(* Logix 5000 project; controller reports 1756-L63 rev 20.11; software revision 20.04; part 38 of 52 *)

        [62].log_data[45].time := 3600.0, [62].log_data[45].valid := 1, [62].log_data[46].time := 3600.0, [62].log_data[46].valid := 1, [62].log_data[47].time := 3600.0, [62].log_data[47].valid := 1, [62].log_data[48].min := 6.623374, [62].log_data[48].max := 6.9811735, [62].log_data[48].total := 24355.637, [62].log_data[48].time := 3600.0, [62].log_data[48].minminute := 59, [62].log_data[48].maxminute := 38, [62].log_data[48].valid := 1, [62].log_data[49].min := 7.172454, [62].log_data[49].max := 9.684395, [62].log_data[49].total := 31171.475, [62].log_data[49].time := 3600.0, [62].log_data[49].minminute := 59, [62].log_data[49].maxminute := 34, [62].log_data[49].valid := 1, [62].log_data[50].min := 2.138653, [62].log_data[50].max := 2.2448862, [62].log_data[50].total := 7885.865, [62].log_data[50].time := 3600.0, [62].log_data[50].minminute := 33, [62].log_data[50].maxminute := 40, [62].log_data[50].valid := 1, [62].log_data[51].time := 3600.0, [62].log_data[51].valid := 1, [62].log_data[52].min := -2.880005, [62].log_data[52].max := 0.11999512, [62].log_data[52].total := -7701.21, [62].log_data[52].time := 3600.0, [62].log_data[52].minminute := 5, [62].log_data[52].maxminute := 3, [62].log_data[52].valid := 1, [62].log_data[53].min := -2.4800034, [62].log_data[53].max := 0.2400055, [62].log_data[53].total := -7366.718, [62].log_data[53].time := 3600.0, [62].log_data[53].maxminute := 40, [62].log_data[53].valid := 1, [62].log_data[54].max := 0.52250004, [62].log_data[54].total := 1217.2524, [62].log_data[54].time := 3600.0, [62].log_data[54].minminute := 3, [62].log_data[54].maxminute := 47, [62].log_data[54].valid := 1, [62].log_data[55].max := 0.5255, [62].log_data[55].total := 1254.6628, [62].log_data[55].time := 3600.0, [62].log_data[55].minminute := 7, [62].log_data[55].maxminute := 19, [62].log_data[55].valid := 1, [62].log_data[56].min := 0.15993154, [62].log_data[56].max := 0.16036338, [62].log_data[56].total := 576.5019, [62].log_data[56].time := 3600.0, [62].log_data[56].minminute := 1, [62].log_data[56].maxminute := 9,
        [62].log_data[56].valid := 1, [62].log_data[57].min := 0.26655704, [62].log_data[57].max := 0.26718515, [62].log_data[57].total := 960.41205, [62].log_data[57].time := 3600.0, [62].log_data[57].minminute := 32, [62].log_data[57].valid := 1, [62].log_data[58].time := 3600.0, [62].log_data[58].valid := 1, [62].log_data[59].time := 3600.0, [62].log_data[59].valid := 1, [62].log_data[60].valid := 1, [62].log_data[61].valid := 1, [62].log_data[62].valid := 1, [62].log_data[63].valid := 1, [62].log_data[64].valid := 1, [62].log_data[65].valid := 1, [62].log_data[66].valid := 1, [62].log_data[67].valid := 1, [62].log_data[68].valid := 1, [62].log_data[69].valid := 1, [62].log_data[70].valid := 1, [62].log_data[71].valid := 1, [62].log_data[72].valid := 1, [62].log_data[73].valid := 1, [62].log_data[74].valid := 1, [62].log_data[75].valid := 1, [62].log_data[76].valid := 1, [62].log_data[77].valid := 1, [62].log_data[78].valid := 1, [62].log_data[79].valid := 1, [62].log_data[80].valid := 1, [62].log_data[81].valid := 1, [62].log_data[82].valid := 1, [62].log_data[83].valid := 1, [62].log_data[84].valid := 1, [62].log_data[85].valid := 1, [62].log_data[86].valid := 1, [62].log_data[87].valid := 1, [62].log_data[88].valid := 1, [62].log_data[89].valid := 1, [62].log_data[90].valid := 1, [62].log_data[91].valid := 1, [62].log_data[92].valid := 1, [62].log_data[93].valid := 1, [62].log_data[94].valid := 1, [62].log_data[95].valid := 1, [62].log_data[96].valid := 1, [62].log_data[97].valid := 1, [62].log_data[98].valid := 1, [62].log_data[99].valid := 1, [62].log_data[100].valid := 1, [62].log_data[101].valid := 1, [62].log_data[102].valid := 1, [62].log_data[103].valid := 1, [62].log_data[104].valid := 1, [62].log_data[105].valid := 1, [62].log_data[106].valid := 1, [62].log_data[107].valid := 1, [62].log_data[108].valid := 1,
        [62].log_data[109].valid := 1, [62].log_data[110].valid := 1, [62].log_data[111].valid := 1, [62].log_data[112].valid := 1, [62].log_data[113].valid := 1, [62].log_data[114].valid := 1, [62].log_data[115].valid := 1, [62].log_data[116].valid := 1, [62].log_data[117].valid := 1, [62].log_data[118].valid := 1, [62].log_data[119].valid := 1, [62].log_data[120].valid := 1, [62].log_data[121].valid := 1, [62].log_data[122].valid := 1, [62].log_data[123].valid := 1, [62].log_data[124].valid := 1, [62].time.Year := 2023, [62].time.Month := 1, [62].time.Day := 15, [62].time.Hour := 17, [62].time.Minute := 59, [62].time.Second := 59, [63].log_data[0].min := 1.0, [63].log_data[0].max := 1.0, [63].log_data[0].total := 3600.0, [63].log_data[0].time := 3600.0, [63].log_data[0].valid := 1, [63].log_data[1].time := 3600.0, [63].log_data[1].valid := 1, [63].log_data[2].time := 3600.0, [63].log_data[2].valid := 1, [63].log_data[3].time := 3600.0, [63].log_data[3].valid := 1, [63].log_data[4].time := 3600.0, [63].log_data[4].valid := 1, [63].log_data[5].time := 3600.0, [63].log_data[5].valid := 1, [63].log_data[6].time := 3600.0, [63].log_data[6].valid := 1, [63].log_data[7].time := 3600.0, [63].log_data[7].valid := 1, [63].log_data[8].min := 1.0, [63].log_data[8].max := 1.0, [63].log_data[8].total := 3600.0, [63].log_data[8].time := 3600.0, [63].log_data[8].valid := 1, [63].log_data[9].min := 1.0, [63].log_data[9].max := 1.0, [63].log_data[9].total := 3600.0, [63].log_data[9].time := 3600.0, [63].log_data[9].valid := 1, [63].log_data[10].min := 1.0, [63].log_data[10].max := 1.0, [63].log_data[10].total := 3600.0, [63].log_data[10].time := 3600.0, [63].log_data[10].valid := 1, [63].log_data[11].time := 3600.0, [63].log_data[11].valid := 1, [63].log_data[12].min := 1.0, [63].log_data[12].max := 1.0,
        [63].log_data[12].total := 3600.0, [63].log_data[12].time := 3600.0, [63].log_data[12].valid := 1, [63].log_data[13].min := 1.0, [63].log_data[13].max := 1.0, [63].log_data[13].total := 3600.0, [63].log_data[13].time := 3600.0, [63].log_data[13].valid := 1, [63].log_data[14].time := 3600.0, [63].log_data[14].valid := 1, [63].log_data[15].time := 3600.0, [63].log_data[15].valid := 1, [63].log_data[16].time := 3600.0, [63].log_data[16].valid := 1, [63].log_data[17].min := 1.0, [63].log_data[17].max := 1.0, [63].log_data[17].total := 3600.0, [63].log_data[17].time := 3600.0, [63].log_data[17].valid := 1, [63].log_data[18].time := 3600.0, [63].log_data[18].valid := 1, [63].log_data[19].time := 3600.0, [63].log_data[19].valid := 1, [63].log_data[20].time := 3600.0, [63].log_data[20].valid := 1, [63].log_data[21].min := 1.0, [63].log_data[21].max := 1.0, [63].log_data[21].total := 3600.0, [63].log_data[21].time := 3600.0, [63].log_data[21].valid := 1, [63].log_data[22].time := 3600.0, [63].log_data[22].valid := 1, [63].log_data[23].time := 3600.0, [63].log_data[23].valid := 1, [63].log_data[24].time := 3600.0, [63].log_data[24].valid := 1, [63].log_data[25].time := 3600.0, [63].log_data[25].valid := 1, [63].log_data[26].time := 3600.0, [63].log_data[26].valid := 1, [63].log_data[27].time := 3600.0, [63].log_data[27].valid := 1, [63].log_data[28].time := 3600.0, [63].log_data[28].valid := 1, [63].log_data[29].min := 1.0, [63].log_data[29].max := 1.0, [63].log_data[29].total := 3600.0, [63].log_data[29].time := 3600.0, [63].log_data[29].valid := 1, [63].log_data[30].min := 1.0, [63].log_data[30].max := 1.0, [63].log_data[30].total := 3600.0, [63].log_data[30].time := 3600.0, [63].log_data[30].valid := 1, [63].log_data[31].max := 1.0, [63].log_data[31].total := 1629.998, [63].log_data[31].time := 3600.0, [63].log_data[31].maxminute := 8, [63].log_data[31].valid := 1, [63].log_data[32].max := 1.0,
        [63].log_data[32].total := 1502.498, [63].log_data[32].time := 3600.0, [63].log_data[32].minminute := 6, [63].log_data[32].valid := 1, [63].log_data[33].time := 3600.0, [63].log_data[33].valid := 1, [63].log_data[34].time := 3600.0, [63].log_data[34].valid := 1, [63].log_data[35].max := 1.0, [63].log_data[35].total := 1440.7471, [63].log_data[35].time := 3600.0, [63].log_data[35].valid := 1, [63].log_data[36].max := 1.0, [63].log_data[36].total := 1629.7471, [63].log_data[36].time := 3600.0, [63].log_data[36].maxminute := 1, [63].log_data[36].valid := 1, [63].log_data[37].time := 3600.0, [63].log_data[37].valid := 1, [63].log_data[38].time := 3600.0, [63].log_data[38].valid := 1, [63].log_data[39].min := 0.99965274, [63].log_data[39].max := 1.0098991, [63].log_data[39].total := 3618.9036, [63].log_data[39].time := 3600.0, [63].log_data[39].minminute := 27, [63].log_data[39].maxminute := 51, [63].log_data[39].valid := 1, [63].log_data[40].min := 7.5689883, [63].log_data[40].max := 7.599217, [63].log_data[40].total := 27323.691, [63].log_data[40].time := 3600.0, [63].log_data[40].minminute := 52, [63].log_data[40].maxminute := 29, [63].log_data[40].valid := 1, [63].log_data[41].min := 0.02273633, [63].log_data[41].max := 0.03628052, [63].log_data[41].total := 100.63758, [63].log_data[41].time := 3600.0, [63].log_data[41].minminute := 33, [63].log_data[41].maxminute := 10, [63].log_data[41].valid := 1, [63].log_data[42].min := 2.2918782, [63].log_data[42].max := 2.2965894, [63].log_data[42].total := 8260.206, [63].log_data[42].time := 3600.0, [63].log_data[42].minminute := 14, [63].log_data[42].maxminute := 40, [63].log_data[42].valid := 1, [63].log_data[43].min := -0.27999878, [63].log_data[43].max := -0.27999878, [63].log_data[43].total := -1007.8613, [63].log_data[43].time := 3600.0, [63].log_data[43].valid := 1, [63].log_data[44].min := -0.3199997, [63].log_data[44].max := -0.30000305, [63].log_data[44].total := -1092.1874, [63].log_data[44].time := 3600.0, [63].log_data[44].valid := 1, [63].log_data[45].time := 3600.0,
        [63].log_data[45].valid := 1, [63].log_data[46].time := 3600.0, [63].log_data[46].valid := 1, [63].log_data[47].time := 3600.0, [63].log_data[47].valid := 1, [63].log_data[48].min := 6.590947, [63].log_data[48].max := 6.7857857, [63].log_data[48].total := 24242.467, [63].log_data[48].time := 3600.0, [63].log_data[48].minminute := 6, [63].log_data[48].maxminute := 19, [63].log_data[48].valid := 1, [63].log_data[49].min := 7.1553764, [63].log_data[49].max := 9.774297, [63].log_data[49].total := 32409.39, [63].log_data[49].time := 3600.0, [63].log_data[49].maxminute := 58, [63].log_data[49].valid := 1, [63].log_data[50].min := 2.1388886, [63].log_data[50].max := 2.2252176, [63].log_data[50].total := 7860.6226, [63].log_data[50].time := 3600.0, [63].log_data[50].minminute := 59, [63].log_data[50].valid := 1, [63].log_data[51].time := 3600.0, [63].log_data[51].valid := 1, [63].log_data[52].min := -2.9000015, [63].log_data[52].max := 0.11999512, [63].log_data[52].total := -7927.2964, [63].log_data[52].time := 3600.0, [63].log_data[52].minminute := 8, [63].log_data[52].maxminute := 7, [63].log_data[52].valid := 1, [63].log_data[53].min := -2.5, [63].log_data[53].max := 0.27999878, [63].log_data[53].total := -7180.0005, [63].log_data[53].time := 3600.0, [63].log_data[53].minminute := 13, [63].log_data[53].maxminute := 1, [63].log_data[53].valid := 1, [63].log_data[54].max := 0.531, [63].log_data[54].total := 1244.2853, [63].log_data[54].time := 3600.0, [63].log_data[54].minminute := 6, [63].log_data[54].maxminute := 29, [63].log_data[54].valid := 1, [63].log_data[55].max := 0.5185, [63].log_data[55].total := 1217.0046, [63].log_data[55].time := 3600.0, [63].log_data[55].maxminute := 54, [63].log_data[55].valid := 1, [63].log_data[56].min := 0.1599708, [63].log_data[56].max := 0.16040264, [63].log_data[56].total := 576.58856, [63].log_data[56].time := 3600.0, [63].log_data[56].minminute := 11, [63].log_data[56].maxminute := 26, [63].log_data[56].valid := 1, [63].log_data[57].min := 0.26534003, [63].log_data[57].max := 0.26694962,
        [63].log_data[57].total := 956.40753, [63].log_data[57].time := 3600.0, [63].log_data[57].minminute := 15, [63].log_data[57].valid := 1, [63].log_data[58].time := 3600.0, [63].log_data[58].valid := 1, [63].log_data[59].time := 3600.0, [63].log_data[59].valid := 1, [63].log_data[60].valid := 1, [63].log_data[61].valid := 1, [63].log_data[62].valid := 1, [63].log_data[63].valid := 1, [63].log_data[64].valid := 1, [63].log_data[65].valid := 1, [63].log_data[66].valid := 1, [63].log_data[67].valid := 1, [63].log_data[68].valid := 1, [63].log_data[69].valid := 1, [63].log_data[70].valid := 1, [63].log_data[71].valid := 1, [63].log_data[72].valid := 1, [63].log_data[73].valid := 1, [63].log_data[74].valid := 1, [63].log_data[75].valid := 1, [63].log_data[76].valid := 1, [63].log_data[77].valid := 1, [63].log_data[78].valid := 1, [63].log_data[79].valid := 1, [63].log_data[80].valid := 1, [63].log_data[81].valid := 1, [63].log_data[82].valid := 1, [63].log_data[83].valid := 1, [63].log_data[84].valid := 1, [63].log_data[85].valid := 1, [63].log_data[86].valid := 1, [63].log_data[87].valid := 1, [63].log_data[88].valid := 1, [63].log_data[89].valid := 1, [63].log_data[90].valid := 1, [63].log_data[91].valid := 1, [63].log_data[92].valid := 1, [63].log_data[93].valid := 1, [63].log_data[94].valid := 1, [63].log_data[95].valid := 1, [63].log_data[96].valid := 1, [63].log_data[97].valid := 1, [63].log_data[98].valid := 1, [63].log_data[99].valid := 1, [63].log_data[100].valid := 1, [63].log_data[101].valid := 1, [63].log_data[102].valid := 1, [63].log_data[103].valid := 1, [63].log_data[104].valid := 1, [63].log_data[105].valid := 1, [63].log_data[106].valid := 1, [63].log_data[107].valid := 1, [63].log_data[108].valid := 1, [63].log_data[109].valid := 1, [63].log_data[110].valid := 1, [63].log_data[111].valid := 1,
        [63].log_data[112].valid := 1, [63].log_data[113].valid := 1, [63].log_data[114].valid := 1, [63].log_data[115].valid := 1, [63].log_data[116].valid := 1, [63].log_data[117].valid := 1, [63].log_data[118].valid := 1, [63].log_data[119].valid := 1, [63].log_data[120].valid := 1, [63].log_data[121].valid := 1, [63].log_data[122].valid := 1, [63].log_data[123].valid := 1, [63].log_data[124].valid := 1, [63].time.Year := 2023, [63].time.Month := 1, [63].time.Day := 15, [63].time.Hour := 18, [63].time.Minute := 59, [63].time.Second := 59, [64].log_data[0].min := 1.0, [64].log_data[0].max := 1.0, [64].log_data[0].total := 3600.0, [64].log_data[0].time := 3600.0, [64].log_data[0].valid := 1, [64].log_data[1].max := 1.0, [64].log_data[1].total := 575.0, [64].log_data[1].time := 3600.0, [64].log_data[1].valid := 1, [64].log_data[2].max := 1.0, [64].log_data[2].total := 571.5, [64].log_data[2].time := 3600.0, [64].log_data[2].valid := 1, [64].log_data[3].time := 3600.0, [64].log_data[3].valid := 1, [64].log_data[4].time := 3600.0, [64].log_data[4].valid := 1, [64].log_data[5].max := 1.0, [64].log_data[5].total := 239.5, [64].log_data[5].time := 3600.0, [64].log_data[5].maxminute := 2, [64].log_data[5].valid := 1, [64].log_data[6].time := 3600.0, [64].log_data[6].valid := 1, [64].log_data[7].time := 3600.0, [64].log_data[7].valid := 1, [64].log_data[8].min := 1.0, [64].log_data[8].max := 1.0, [64].log_data[8].total := 3600.0, [64].log_data[8].time := 3600.0, [64].log_data[8].valid := 1, [64].log_data[9].min := 1.0, [64].log_data[9].max := 1.0, [64].log_data[9].total := 3600.0, [64].log_data[9].time := 3600.0, [64].log_data[9].valid := 1, [64].log_data[10].min := 1.0, [64].log_data[10].max := 1.0, [64].log_data[10].total := 3600.0, [64].log_data[10].time := 3600.0, [64].log_data[10].valid := 1,
        [64].log_data[11].time := 3600.0, [64].log_data[11].valid := 1, [64].log_data[12].min := 1.0, [64].log_data[12].max := 1.0, [64].log_data[12].total := 3600.0, [64].log_data[12].time := 3600.0, [64].log_data[12].valid := 1, [64].log_data[13].min := 1.0, [64].log_data[13].max := 1.0, [64].log_data[13].total := 3600.0, [64].log_data[13].time := 3600.0, [64].log_data[13].valid := 1, [64].log_data[14].time := 3600.0, [64].log_data[14].valid := 1, [64].log_data[15].time := 3600.0, [64].log_data[15].valid := 1, [64].log_data[16].time := 3600.0, [64].log_data[16].valid := 1, [64].log_data[17].min := 1.0, [64].log_data[17].max := 1.0, [64].log_data[17].total := 3600.0, [64].log_data[17].time := 3600.0, [64].log_data[17].valid := 1, [64].log_data[18].time := 3600.0, [64].log_data[18].valid := 1, [64].log_data[19].time := 3600.0, [64].log_data[19].valid := 1, [64].log_data[20].time := 3600.0, [64].log_data[20].valid := 1, [64].log_data[21].min := 1.0, [64].log_data[21].max := 1.0, [64].log_data[21].total := 3600.0, [64].log_data[21].time := 3600.0, [64].log_data[21].valid := 1, [64].log_data[22].time := 3600.0, [64].log_data[22].valid := 1, [64].log_data[23].time := 3600.0, [64].log_data[23].valid := 1, [64].log_data[24].time := 3600.0, [64].log_data[24].valid := 1, [64].log_data[25].time := 3600.0, [64].log_data[25].valid := 1, [64].log_data[26].time := 3600.0, [64].log_data[26].valid := 1, [64].log_data[27].time := 3600.0, [64].log_data[27].valid := 1, [64].log_data[28].time := 3600.0, [64].log_data[28].valid := 1, [64].log_data[29].min := 1.0, [64].log_data[29].max := 1.0, [64].log_data[29].total := 3600.0, [64].log_data[29].time := 3600.0, [64].log_data[29].valid := 1, [64].log_data[30].min := 1.0, [64].log_data[30].max := 1.0, [64].log_data[30].total := 3600.0, [64].log_data[30].time := 3600.0, [64].log_data[30].valid := 1, [64].log_data[31].max := 1.0, [64].log_data[31].total := 1467.2471,
        [64].log_data[31].time := 3600.0, [64].log_data[31].maxminute := 11, [64].log_data[31].valid := 1, [64].log_data[32].max := 1.0, [64].log_data[32].total := 1629.7471, [64].log_data[32].time := 3600.0, [64].log_data[32].maxminute := 1, [64].log_data[32].valid := 1, [64].log_data[33].time := 3600.0, [64].log_data[33].valid := 1, [64].log_data[34].time := 3600.0, [64].log_data[34].valid := 1, [64].log_data[35].max := 1.0, [64].log_data[35].total := 1440.7471, [64].log_data[35].time := 3600.0, [64].log_data[35].minminute := 3, [64].log_data[35].valid := 1, [64].log_data[36].max := 1.0, [64].log_data[36].total := 1629.7471, [64].log_data[36].time := 3600.0, [64].log_data[36].maxminute := 5, [64].log_data[36].valid := 1, [64].log_data[37].max := 7.22856, [64].log_data[37].total := 3622.7856, [64].log_data[37].time := 3600.0, [64].log_data[37].maxminute := 1, [64].log_data[37].valid := 1, [64].log_data[38].time := 3600.0, [64].log_data[38].valid := 1, [64].log_data[39].min := 0.9982394, [64].log_data[39].max := 1.02203, [64].log_data[39].total := 3625.5354, [64].log_data[39].time := 3600.0, [64].log_data[39].minminute := 8, [64].log_data[39].maxminute := 6, [64].log_data[39].valid := 1, [64].log_data[40].min := 7.560194, [64].log_data[40].max := 7.6063623, [64].log_data[40].total := 27324.1, [64].log_data[40].time := 3600.0, [64].log_data[40].minminute := 56, [64].log_data[40].maxminute := 59, [64].log_data[40].valid := 1, [64].log_data[41].min := 0.025877198, [64].log_data[41].max := 0.044524662, [64].log_data[41].total := 125.660706, [64].log_data[41].time := 3600.0, [64].log_data[41].maxminute := 30, [64].log_data[41].valid := 1, [64].log_data[42].min := 2.2917604, [64].log_data[42].max := 2.2964714, [64].log_data[42].total := 8260.182, [64].log_data[42].time := 3600.0, [64].log_data[42].minminute := 28, [64].log_data[42].maxminute := 24, [64].log_data[42].valid := 1, [64].log_data[43].min := -0.27999878, [64].log_data[43].max := -0.26000214, [64].log_data[43].total := -1007.73706, [64].log_data[43].time := 3600.0,
        [64].log_data[43].maxminute := 9, [64].log_data[43].valid := 1, [64].log_data[44].min := -0.3199997, [64].log_data[44].max := -0.30000305, [64].log_data[44].total := -1087.6062, [64].log_data[44].time := 3600.0, [64].log_data[44].valid := 1, [64].log_data[45].time := 3600.0, [64].log_data[45].valid := 1, [64].log_data[46].time := 3600.0, [64].log_data[46].valid := 1, [64].log_data[47].time := 3600.0, [64].log_data[47].valid := 1, [64].log_data[48].min := 6.588199, [64].log_data[48].max := 6.952594, [64].log_data[48].total := 24228.959, [64].log_data[48].time := 3600.0, [64].log_data[48].minminute := 33, [64].log_data[48].maxminute := 3, [64].log_data[48].valid := 1, [64].log_data[49].min := 7.1818757, [64].log_data[49].max := 9.775277, [64].log_data[49].total := 29847.389, [64].log_data[49].time := 3600.0, [64].log_data[49].minminute := 30, [64].log_data[49].maxminute := 1, [64].log_data[49].valid := 1, [64].log_data[50].min := 2.13512, [64].log_data[50].max := 2.2438262, [64].log_data[50].total := 7948.6934, [64].log_data[50].time := 3600.0, [64].log_data[50].minminute := 1, [64].log_data[50].maxminute := 11, [64].log_data[50].valid := 1, [64].log_data[51].time := 3600.0, [64].log_data[51].valid := 1, [64].log_data[52].min := -2.959999, [64].log_data[52].max := 0.11999512, [64].log_data[52].total := -7812.1035, [64].log_data[52].time := 3600.0, [64].log_data[52].minminute := 11, [64].log_data[52].valid := 1, [64].log_data[53].min := -2.600006, [64].log_data[53].max := 0.2400055, [64].log_data[53].total := -7210.3994, [64].log_data[53].time := 3600.0, [64].log_data[53].minminute := 15, [64].log_data[53].maxminute := 25, [64].log_data[53].valid := 1, [64].log_data[54].max := 0.54, [64].log_data[54].total := 1227.2667, [64].log_data[54].time := 3600.0, [64].log_data[54].maxminute := 11, [64].log_data[54].valid := 1, [64].log_data[55].max := 0.539, [64].log_data[55].total := 1217.0822, [64].log_data[55].time := 3600.0, [64].log_data[55].minminute := 3, [64].log_data[55].maxminute := 57, [64].log_data[55].valid := 1,
        [64].log_data[56].min := 0.16001005, [64].log_data[56].max := 0.16044189, [64].log_data[56].total := 576.6807, [64].log_data[56].time := 3600.0, [64].log_data[56].minminute := 32, [64].log_data[56].maxminute := 29, [64].log_data[56].valid := 1, [64].log_data[57].min := 0.26380894, [64].log_data[57].max := 0.26569337, [64].log_data[57].total := 953.66, [64].log_data[57].time := 3600.0, [64].log_data[57].minminute := 50, [64].log_data[57].maxminute := 6, [64].log_data[57].valid := 1, [64].log_data[58].time := 3600.0, [64].log_data[58].valid := 1, [64].log_data[59].time := 3600.0, [64].log_data[59].valid := 1, [64].log_data[60].valid := 1, [64].log_data[61].valid := 1, [64].log_data[62].valid := 1, [64].log_data[63].valid := 1, [64].log_data[64].valid := 1, [64].log_data[65].valid := 1, [64].log_data[66].valid := 1, [64].log_data[67].valid := 1, [64].log_data[68].valid := 1, [64].log_data[69].valid := 1, [64].log_data[70].valid := 1, [64].log_data[71].valid := 1, [64].log_data[72].valid := 1, [64].log_data[73].valid := 1, [64].log_data[74].valid := 1, [64].log_data[75].valid := 1, [64].log_data[76].valid := 1, [64].log_data[77].valid := 1, [64].log_data[78].valid := 1, [64].log_data[79].valid := 1, [64].log_data[80].valid := 1, [64].log_data[81].valid := 1, [64].log_data[82].valid := 1, [64].log_data[83].valid := 1, [64].log_data[84].valid := 1, [64].log_data[85].valid := 1, [64].log_data[86].valid := 1, [64].log_data[87].valid := 1, [64].log_data[88].valid := 1, [64].log_data[89].valid := 1, [64].log_data[90].valid := 1, [64].log_data[91].valid := 1, [64].log_data[92].valid := 1, [64].log_data[93].valid := 1, [64].log_data[94].valid := 1, [64].log_data[95].valid := 1, [64].log_data[96].valid := 1, [64].log_data[97].valid := 1, [64].log_data[98].valid := 1, [64].log_data[99].valid := 1, [64].log_data[100].valid := 1, [64].log_data[101].valid := 1,
        [64].log_data[102].valid := 1, [64].log_data[103].valid := 1, [64].log_data[104].valid := 1, [64].log_data[105].valid := 1, [64].log_data[106].valid := 1, [64].log_data[107].valid := 1, [64].log_data[108].valid := 1, [64].log_data[109].valid := 1, [64].log_data[110].valid := 1, [64].log_data[111].valid := 1, [64].log_data[112].valid := 1, [64].log_data[113].valid := 1, [64].log_data[114].valid := 1, [64].log_data[115].valid := 1, [64].log_data[116].valid := 1, [64].log_data[117].valid := 1, [64].log_data[118].valid := 1, [64].log_data[119].valid := 1, [64].log_data[120].valid := 1, [64].log_data[121].valid := 1, [64].log_data[122].valid := 1, [64].log_data[123].valid := 1, [64].log_data[124].valid := 1, [64].time.Year := 2023, [64].time.Month := 1, [64].time.Day := 15, [64].time.Hour := 19, [64].time.Minute := 59, [64].time.Second := 59, [65].log_data[0].min := 1.0, [65].log_data[0].max := 1.0, [65].log_data[0].total := 3600.0, [65].log_data[0].time := 3600.0, [65].log_data[0].valid := 1, [65].log_data[1].max := 1.0, [65].log_data[1].total := 552.0, [65].log_data[1].time := 3600.0, [65].log_data[1].maxminute := 8, [65].log_data[1].valid := 1, [65].log_data[2].max := 1.0, [65].log_data[2].total := 548.5, [65].log_data[2].time := 3600.0, [65].log_data[2].maxminute := 8, [65].log_data[2].valid := 1, [65].log_data[3].time := 3600.0, [65].log_data[3].valid := 1, [65].log_data[4].time := 3600.0, [65].log_data[4].valid := 1, [65].log_data[5].max := 1.0, [65].log_data[5].total := 250.5, [65].log_data[5].time := 3600.0, [65].log_data[5].maxminute := 10, [65].log_data[5].valid := 1, [65].log_data[6].time := 3600.0, [65].log_data[6].valid := 1, [65].log_data[7].time := 3600.0, [65].log_data[7].valid := 1, [65].log_data[8].min := 1.0, [65].log_data[8].max := 1.0, [65].log_data[8].total := 3600.0,
        [65].log_data[8].time := 3600.0, [65].log_data[8].valid := 1, [65].log_data[9].min := 1.0, [65].log_data[9].max := 1.0, [65].log_data[9].total := 3600.0, [65].log_data[9].time := 3600.0, [65].log_data[9].valid := 1, [65].log_data[10].min := 1.0, [65].log_data[10].max := 1.0, [65].log_data[10].total := 3600.0, [65].log_data[10].time := 3600.0, [65].log_data[10].valid := 1, [65].log_data[11].time := 3600.0, [65].log_data[11].valid := 1, [65].log_data[12].min := 1.0, [65].log_data[12].max := 1.0, [65].log_data[12].total := 3600.0, [65].log_data[12].time := 3600.0, [65].log_data[12].valid := 1, [65].log_data[13].min := 1.0, [65].log_data[13].max := 1.0, [65].log_data[13].total := 3600.0, [65].log_data[13].time := 3600.0, [65].log_data[13].valid := 1, [65].log_data[14].time := 3600.0, [65].log_data[14].valid := 1, [65].log_data[15].time := 3600.0, [65].log_data[15].valid := 1, [65].log_data[16].time := 3600.0, [65].log_data[16].valid := 1, [65].log_data[17].min := 1.0, [65].log_data[17].max := 1.0, [65].log_data[17].total := 3600.0, [65].log_data[17].time := 3600.0, [65].log_data[17].valid := 1, [65].log_data[18].time := 3600.0, [65].log_data[18].valid := 1, [65].log_data[19].time := 3600.0, [65].log_data[19].valid := 1, [65].log_data[20].time := 3600.0, [65].log_data[20].valid := 1, [65].log_data[21].min := 1.0, [65].log_data[21].max := 1.0, [65].log_data[21].total := 3600.0, [65].log_data[21].time := 3600.0, [65].log_data[21].valid := 1, [65].log_data[22].time := 3600.0, [65].log_data[22].valid := 1, [65].log_data[23].time := 3600.0, [65].log_data[23].valid := 1, [65].log_data[24].time := 3600.0, [65].log_data[24].valid := 1, [65].log_data[25].time := 3600.0, [65].log_data[25].valid := 1, [65].log_data[26].time := 3600.0, [65].log_data[26].valid := 1, [65].log_data[27].time := 3600.0, [65].log_data[27].valid := 1, [65].log_data[28].time := 3600.0, [65].log_data[28].valid := 1,
        [65].log_data[29].min := 1.0, [65].log_data[29].max := 1.0, [65].log_data[29].total := 3600.0, [65].log_data[29].time := 3600.0, [65].log_data[29].valid := 1, [65].log_data[30].min := 1.0, [65].log_data[30].max := 1.0, [65].log_data[30].total := 3600.0, [65].log_data[30].time := 3600.0, [65].log_data[30].valid := 1, [65].log_data[31].max := 1.0, [65].log_data[31].total := 1441.249, [65].log_data[31].time := 3600.0, [65].log_data[31].minminute := 2, [65].log_data[31].valid := 1, [65].log_data[32].max := 1.0, [65].log_data[32].total := 1629.749, [65].log_data[32].time := 3600.0, [65].log_data[32].maxminute := 4, [65].log_data[32].valid := 1, [65].log_data[33].time := 3600.0, [65].log_data[33].valid := 1, [65].log_data[34].time := 3600.0, [65].log_data[34].valid := 1, [65].log_data[35].max := 1.0, [65].log_data[35].total := 1491.998, [65].log_data[35].time := 3600.0, [65].log_data[35].minminute := 6, [65].log_data[35].valid := 1, [65].log_data[36].max := 1.0, [65].log_data[36].total := 1629.998, [65].log_data[36].time := 3600.0, [65].log_data[36].maxminute := 8, [65].log_data[36].valid := 1, [65].log_data[37].max := 7.450369, [65].log_data[37].total := 3580.0767, [65].log_data[37].time := 3600.0, [65].log_data[37].maxminute := 9, [65].log_data[37].valid := 1, [65].log_data[38].time := 3600.0, [65].log_data[38].valid := 1, [65].log_data[39].min := 0.99800396, [65].log_data[39].max := 1.0223833, [65].log_data[39].total := 3620.6714, [65].log_data[39].time := 3600.0, [65].log_data[39].minminute := 59, [65].log_data[39].maxminute := 10, [65].log_data[39].valid := 1, [65].log_data[40].min := 7.557446, [65].log_data[40].max := 7.611859, [65].log_data[40].total := 27325.555, [65].log_data[40].time := 3600.0, [65].log_data[40].minminute := 37, [65].log_data[40].maxminute := 40, [65].log_data[40].valid := 1, [65].log_data[41].min := 0.02273633, [65].log_data[41].max := 0.034317628, [65].log_data[41].total := 96.31372, [65].log_data[41].time := 3600.0, [65].log_data[41].minminute := 29,
        [65].log_data[41].maxminute := 7, [65].log_data[41].valid := 1, [65].log_data[42].min := 2.291996, [65].log_data[42].max := 2.2968247, [65].log_data[42].total := 8260.134, [65].log_data[42].time := 3600.0, [65].log_data[42].minminute := 40, [65].log_data[42].maxminute := 35, [65].log_data[42].valid := 1, [65].log_data[43].min := -0.27999878, [65].log_data[43].max := -0.26000214, [65].log_data[43].total := -1007.21295, [65].log_data[43].time := 3600.0, [65].log_data[43].maxminute := 9, [65].log_data[43].valid := 1, [65].log_data[44].min := -0.3199997, [65].log_data[44].max := -0.30000305, [65].log_data[44].total := -1082.1633, [65].log_data[44].time := 3600.0, [65].log_data[44].valid := 1, [65].log_data[45].time := 3600.0, [65].log_data[45].valid := 1, [65].log_data[46].time := 3600.0, [65].log_data[46].valid := 1, [65].log_data[47].time := 3600.0, [65].log_data[47].valid := 1, [65].log_data[48].min := 6.5824285, [65].log_data[48].max := 6.969357, [65].log_data[48].total := 24224.227, [65].log_data[48].time := 3600.0, [65].log_data[48].minminute := 42, [65].log_data[48].maxminute := 17, [65].log_data[48].valid := 1, [65].log_data[49].min := 7.0841227, [65].log_data[49].max := 9.659073, [65].log_data[49].total := 29661.438, [65].log_data[49].time := 3600.0, [65].log_data[49].minminute := 39, [65].log_data[49].maxminute := 10, [65].log_data[49].valid := 1, [65].log_data[50].min := 2.163268, [65].log_data[50].max := 2.276332, [65].log_data[50].total := 8044.48, [65].log_data[50].time := 3600.0, [65].log_data[50].minminute := 10, [65].log_data[50].maxminute := 18, [65].log_data[50].valid := 1, [65].log_data[51].time := 3600.0, [65].log_data[51].valid := 1, [65].log_data[52].min := -2.959999, [65].log_data[52].max := 0.11999512, [65].log_data[52].total := -7730.7188, [65].log_data[52].time := 3600.0, [65].log_data[52].minminute := 56, [65].log_data[52].maxminute := 2, [65].log_data[52].valid := 1, [65].log_data[53].min := -2.6600037, [65].log_data[53].max := 0.27999878, [65].log_data[53].total := -7362.1255, [65].log_data[53].time := 3600.0,
        [65].log_data[53].minminute := 8, [65].log_data[53].maxminute := 7, [65].log_data[53].valid := 1, [65].log_data[54].max := 0.53, [65].log_data[54].total := 1217.8265, [65].log_data[54].time := 3600.0, [65].log_data[54].minminute := 2, [65].log_data[54].maxminute := 56, [65].log_data[54].valid := 1, [65].log_data[55].max := 0.546, [65].log_data[55].total := 1240.171, [65].log_data[55].time := 3600.0, [65].log_data[55].minminute := 6, [65].log_data[55].maxminute := 18, [65].log_data[55].valid := 1, [65].log_data[56].min := 0.16001005, [65].log_data[56].max := 0.16044189, [65].log_data[56].total := 576.7335, [65].log_data[56].time := 3600.0, [65].log_data[56].minminute := 39, [65].log_data[56].maxminute := 14, [65].log_data[56].valid := 1, [65].log_data[57].min := 0.2618068, [65].log_data[57].max := 0.26424077, [65].log_data[57].total := 948.47955, [65].log_data[57].time := 3600.0, [65].log_data[57].minminute := 58, [65].log_data[57].maxminute := 13, [65].log_data[57].valid := 1, [65].log_data[58].time := 3600.0, [65].log_data[58].valid := 1, [65].log_data[59].time := 3600.0, [65].log_data[59].valid := 1, [65].log_data[60].valid := 1, [65].log_data[61].valid := 1, [65].log_data[62].valid := 1, [65].log_data[63].valid := 1, [65].log_data[64].valid := 1, [65].log_data[65].valid := 1, [65].log_data[66].valid := 1, [65].log_data[67].valid := 1, [65].log_data[68].valid := 1, [65].log_data[69].valid := 1, [65].log_data[70].valid := 1, [65].log_data[71].valid := 1, [65].log_data[72].valid := 1, [65].log_data[73].valid := 1, [65].log_data[74].valid := 1, [65].log_data[75].valid := 1, [65].log_data[76].valid := 1, [65].log_data[77].valid := 1, [65].log_data[78].valid := 1, [65].log_data[79].valid := 1, [65].log_data[80].valid := 1, [65].log_data[81].valid := 1, [65].log_data[82].valid := 1, [65].log_data[83].valid := 1, [65].log_data[84].valid := 1, [65].log_data[85].valid := 1, [65].log_data[86].valid := 1,
        [65].log_data[87].valid := 1, [65].log_data[88].valid := 1, [65].log_data[89].valid := 1, [65].log_data[90].valid := 1, [65].log_data[91].valid := 1, [65].log_data[92].valid := 1, [65].log_data[93].valid := 1, [65].log_data[94].valid := 1, [65].log_data[95].valid := 1, [65].log_data[96].valid := 1, [65].log_data[97].valid := 1, [65].log_data[98].valid := 1, [65].log_data[99].valid := 1, [65].log_data[100].valid := 1, [65].log_data[101].valid := 1, [65].log_data[102].valid := 1, [65].log_data[103].valid := 1, [65].log_data[104].valid := 1, [65].log_data[105].valid := 1, [65].log_data[106].valid := 1, [65].log_data[107].valid := 1, [65].log_data[108].valid := 1, [65].log_data[109].valid := 1, [65].log_data[110].valid := 1, [65].log_data[111].valid := 1, [65].log_data[112].valid := 1, [65].log_data[113].valid := 1, [65].log_data[114].valid := 1, [65].log_data[115].valid := 1, [65].log_data[116].valid := 1, [65].log_data[117].valid := 1, [65].log_data[118].valid := 1, [65].log_data[119].valid := 1, [65].log_data[120].valid := 1, [65].log_data[121].valid := 1, [65].log_data[122].valid := 1, [65].log_data[123].valid := 1, [65].log_data[124].valid := 1, [65].time.Year := 2023, [65].time.Month := 1, [65].time.Day := 15, [65].time.Hour := 20, [65].time.Minute := 59, [65].time.Second := 59, [66].log_data[0].min := 1.0, [66].log_data[0].max := 1.0, [66].log_data[0].total := 3600.0, [66].log_data[0].time := 3600.0, [66].log_data[0].valid := 1, [66].log_data[1].max := 1.0, [66].log_data[1].total := 570.5, [66].log_data[1].time := 3600.0, [66].log_data[1].maxminute := 22, [66].log_data[1].valid := 1, [66].log_data[2].max := 1.0, [66].log_data[2].total := 567.0, [66].log_data[2].time := 3600.0, [66].log_data[2].maxminute := 22, [66].log_data[2].valid := 1, [66].log_data[3].time := 3600.0,
        [66].log_data[3].valid := 1, [66].log_data[4].time := 3600.0, [66].log_data[4].valid := 1, [66].log_data[5].max := 1.0, [66].log_data[5].total := 233.5, [66].log_data[5].time := 3600.0, [66].log_data[5].maxminute := 24, [66].log_data[5].valid := 1, [66].log_data[6].time := 3600.0, [66].log_data[6].valid := 1, [66].log_data[7].time := 3600.0, [66].log_data[7].valid := 1, [66].log_data[8].min := 1.0, [66].log_data[8].max := 1.0, [66].log_data[8].total := 3600.0, [66].log_data[8].time := 3600.0, [66].log_data[8].valid := 1, [66].log_data[9].min := 1.0, [66].log_data[9].max := 1.0, [66].log_data[9].total := 3600.0, [66].log_data[9].time := 3600.0, [66].log_data[9].valid := 1, [66].log_data[10].min := 1.0, [66].log_data[10].max := 1.0, [66].log_data[10].total := 3600.0, [66].log_data[10].time := 3600.0, [66].log_data[10].valid := 1, [66].log_data[11].time := 3600.0, [66].log_data[11].valid := 1, [66].log_data[12].min := 1.0, [66].log_data[12].max := 1.0, [66].log_data[12].total := 3600.0, [66].log_data[12].time := 3600.0, [66].log_data[12].valid := 1, [66].log_data[13].min := 1.0, [66].log_data[13].max := 1.0, [66].log_data[13].total := 3600.0, [66].log_data[13].time := 3600.0, [66].log_data[13].valid := 1, [66].log_data[14].time := 3600.0, [66].log_data[14].valid := 1, [66].log_data[15].time := 3600.0, [66].log_data[15].valid := 1, [66].log_data[16].time := 3600.0, [66].log_data[16].valid := 1, [66].log_data[17].min := 1.0, [66].log_data[17].max := 1.0, [66].log_data[17].total := 3600.0, [66].log_data[17].time := 3600.0, [66].log_data[17].valid := 1, [66].log_data[18].time := 3600.0, [66].log_data[18].valid := 1, [66].log_data[19].time := 3600.0, [66].log_data[19].valid := 1, [66].log_data[20].time := 3600.0, [66].log_data[20].valid := 1, [66].log_data[21].min := 1.0, [66].log_data[21].max := 1.0, [66].log_data[21].total := 3600.0, [66].log_data[21].time := 3600.0,
        [66].log_data[21].valid := 1, [66].log_data[22].time := 3600.0, [66].log_data[22].valid := 1, [66].log_data[23].time := 3600.0, [66].log_data[23].valid := 1, [66].log_data[24].time := 3600.0, [66].log_data[24].valid := 1, [66].log_data[25].time := 3600.0, [66].log_data[25].valid := 1, [66].log_data[26].time := 3600.0, [66].log_data[26].valid := 1, [66].log_data[27].time := 3600.0, [66].log_data[27].valid := 1, [66].log_data[28].time := 3600.0, [66].log_data[28].valid := 1, [66].log_data[29].min := 1.0, [66].log_data[29].max := 1.0, [66].log_data[29].total := 3600.0, [66].log_data[29].time := 3600.0, [66].log_data[29].valid := 1, [66].log_data[30].min := 1.0, [66].log_data[30].max := 1.0, [66].log_data[30].total := 3600.0, [66].log_data[30].time := 3600.0, [66].log_data[30].valid := 1, [66].log_data[31].max := 1.0, [66].log_data[31].total := 1440.7471, [66].log_data[31].time := 3600.0, [66].log_data[31].minminute := 5, [66].log_data[31].valid := 1, [66].log_data[32].max := 1.0, [66].log_data[32].total := 1629.7471, [66].log_data[32].time := 3600.0, [66].log_data[32].maxminute := 7, [66].log_data[32].valid := 1, [66].log_data[33].time := 3600.0, [66].log_data[33].valid := 1, [66].log_data[34].time := 3600.0, [66].log_data[34].valid := 1, [66].log_data[35].max := 1.0, [66].log_data[35].total := 1629.7471, [66].log_data[35].time := 3600.0, [66].log_data[35].valid := 1, [66].log_data[36].max := 1.0, [66].log_data[36].total := 1477.2471, [66].log_data[36].time := 3600.0, [66].log_data[36].maxminute := 11, [66].log_data[36].valid := 1, [66].log_data[37].max := 7.21796, [66].log_data[37].total := 3591.0007, [66].log_data[37].time := 3600.0, [66].log_data[37].maxminute := 23, [66].log_data[37].valid := 1, [66].log_data[38].time := 3600.0, [66].log_data[38].valid := 1, [66].log_data[39].min := 0.99776834, [66].log_data[39].max := 1.0212055, [66].log_data[39].total := 3622.2793, [66].log_data[39].time := 3600.0, [66].log_data[39].minminute := 26,
        [66].log_data[39].maxminute := 28, [66].log_data[39].valid := 1, [66].log_data[40].min := 7.5700884, [66].log_data[40].max := 7.598118, [66].log_data[40].total := 27323.703, [66].log_data[40].time := 3600.0, [66].log_data[40].minminute := 9, [66].log_data[40].maxminute := 2, [66].log_data[40].valid := 1, [66].log_data[41].min := 0.02273633, [66].log_data[41].max := 0.028232668, [66].log_data[41].total := 87.084, [66].log_data[41].time := 3600.0, [66].log_data[41].maxminute := 50, [66].log_data[41].valid := 1, [66].log_data[42].min := 2.291525, [66].log_data[42].max := 2.2964714, [66].log_data[42].total := 8260.155, [66].log_data[42].time := 3600.0, [66].log_data[42].minminute := 20, [66].log_data[42].maxminute := 56, [66].log_data[42].valid := 1, [66].log_data[43].min := -0.27999878, [66].log_data[43].max := -0.26000214, [66].log_data[43].total := -993.043, [66].log_data[43].time := 3600.0, [66].log_data[43].valid := 1, [66].log_data[44].min := -0.3199997, [66].log_data[44].max := -0.30000305, [66].log_data[44].total := -1080.1062, [66].log_data[44].time := 3600.0, [66].log_data[44].minminute := 14, [66].log_data[44].valid := 1, [66].log_data[45].time := 3600.0, [66].log_data[45].valid := 1, [66].log_data[46].time := 3600.0, [66].log_data[46].valid := 1, [66].log_data[47].time := 3600.0, [66].log_data[47].valid := 1, [66].log_data[48].min := 6.595344, [66].log_data[48].max := 6.959464, [66].log_data[48].total := 24285.668, [66].log_data[48].time := 3600.0, [66].log_data[48].minminute := 57, [66].log_data[48].maxminute := 26, [66].log_data[48].valid := 1, [66].log_data[49].min := 7.1871758, [66].log_data[49].max := 9.70108, [66].log_data[49].total := 30726.588, [66].log_data[49].time := 3600.0, [66].log_data[49].minminute := 47, [66].log_data[49].maxminute := 24, [66].log_data[49].valid := 1, [66].log_data[50].min := 2.188943, [66].log_data[50].max := 2.292467, [66].log_data[50].total := 8078.358, [66].log_data[50].time := 3600.0, [66].log_data[50].minminute := 24, [66].log_data[50].maxminute := 34, [66].log_data[50].valid := 1,
        [66].log_data[51].time := 3600.0, [66].log_data[51].valid := 1, [66].log_data[52].min := -3.0599976, [66].log_data[52].max := 0.11999512, [66].log_data[52].total := -7782.3887, [66].log_data[52].time := 3600.0, [66].log_data[52].minminute := 17, [66].log_data[52].maxminute := 5, [66].log_data[52].valid := 1, [66].log_data[53].min := -2.7000046, [66].log_data[53].max := 0.27999878, [66].log_data[53].total := -7383.723, [66].log_data[53].time := 3600.0, [66].log_data[53].minminute := 21, [66].log_data[53].maxminute := 42, [66].log_data[53].valid := 1, [66].log_data[54].max := 0.5465, [66].log_data[54].total := 1218.1571, [66].log_data[54].time := 3600.0, [66].log_data[54].minminute := 5, [66].log_data[54].maxminute := 17, [66].log_data[54].valid := 1, [66].log_data[55].max := 0.55050004, [66].log_data[55].total := 1231.6753, [66].log_data[55].time := 3600.0, [66].log_data[55].maxminute := 22, [66].log_data[55].valid := 1, [66].log_data[56].min := 0.16008857, [66].log_data[56].max := 0.16048115, [66].log_data[56].total := 576.91205, [66].log_data[56].time := 3600.0, [66].log_data[56].minminute := 58, [66].log_data[56].maxminute := 1, [66].log_data[56].valid := 1, [66].log_data[57].min := 0.26117867, [66].log_data[57].max := 0.26227787, [66].log_data[57].total := 943.17426, [66].log_data[57].time := 3600.0, [66].log_data[57].minminute := 59, [66].log_data[57].maxminute := 37, [66].log_data[57].valid := 1, [66].log_data[58].time := 3600.0, [66].log_data[58].valid := 1, [66].log_data[59].time := 3600.0, [66].log_data[59].valid := 1, [66].log_data[60].valid := 1, [66].log_data[61].valid := 1, [66].log_data[62].valid := 1, [66].log_data[63].valid := 1, [66].log_data[64].valid := 1, [66].log_data[65].valid := 1, [66].log_data[66].valid := 1, [66].log_data[67].valid := 1, [66].log_data[68].valid := 1, [66].log_data[69].valid := 1, [66].log_data[70].valid := 1, [66].log_data[71].valid := 1, [66].log_data[72].valid := 1, [66].log_data[73].valid := 1, [66].log_data[74].valid := 1,
        [66].log_data[75].valid := 1, [66].log_data[76].valid := 1, [66].log_data[77].valid := 1, [66].log_data[78].valid := 1, [66].log_data[79].valid := 1, [66].log_data[80].valid := 1, [66].log_data[81].valid := 1, [66].log_data[82].valid := 1, [66].log_data[83].valid := 1, [66].log_data[84].valid := 1, [66].log_data[85].valid := 1, [66].log_data[86].valid := 1, [66].log_data[87].valid := 1, [66].log_data[88].valid := 1, [66].log_data[89].valid := 1, [66].log_data[90].valid := 1, [66].log_data[91].valid := 1, [66].log_data[92].valid := 1, [66].log_data[93].valid := 1, [66].log_data[94].valid := 1, [66].log_data[95].valid := 1, [66].log_data[96].valid := 1, [66].log_data[97].valid := 1, [66].log_data[98].valid := 1, [66].log_data[99].valid := 1, [66].log_data[100].valid := 1, [66].log_data[101].valid := 1, [66].log_data[102].valid := 1, [66].log_data[103].valid := 1, [66].log_data[104].valid := 1, [66].log_data[105].valid := 1, [66].log_data[106].valid := 1, [66].log_data[107].valid := 1, [66].log_data[108].valid := 1, [66].log_data[109].valid := 1, [66].log_data[110].valid := 1, [66].log_data[111].valid := 1, [66].log_data[112].valid := 1, [66].log_data[113].valid := 1, [66].log_data[114].valid := 1, [66].log_data[115].valid := 1, [66].log_data[116].valid := 1, [66].log_data[117].valid := 1, [66].log_data[118].valid := 1, [66].log_data[119].valid := 1, [66].log_data[120].valid := 1, [66].log_data[121].valid := 1, [66].log_data[122].valid := 1, [66].log_data[123].valid := 1, [66].log_data[124].valid := 1, [66].time.Year := 2023, [66].time.Month := 1, [66].time.Day := 15, [66].time.Hour := 21, [66].time.Minute := 59, [66].time.Second := 59, [67].log_data[0].min := 1.0, [67].log_data[0].max := 1.0, [67].log_data[0].total := 3599.5, [67].log_data[0].time := 3599.5,
        [67].log_data[0].valid := 1, [67].log_data[1].max := 1.0, [67].log_data[1].total := 541.5, [67].log_data[1].time := 3599.5, [67].log_data[1].maxminute := 42, [67].log_data[1].valid := 1, [67].log_data[2].max := 1.0, [67].log_data[2].total := 538.0, [67].log_data[2].time := 3599.5, [67].log_data[2].maxminute := 42, [67].log_data[2].valid := 1, [67].log_data[3].time := 3599.5, [67].log_data[3].valid := 1, [67].log_data[4].time := 3599.5, [67].log_data[4].valid := 1, [67].log_data[5].max := 1.0, [67].log_data[5].total := 244.5, [67].log_data[5].time := 3599.5, [67].log_data[5].maxminute := 43, [67].log_data[5].valid := 1, [67].log_data[6].time := 3599.5, [67].log_data[6].valid := 1, [67].log_data[7].time := 3599.5, [67].log_data[7].valid := 1, [67].log_data[8].min := 1.0, [67].log_data[8].max := 1.0, [67].log_data[8].total := 3599.5, [67].log_data[8].time := 3599.5, [67].log_data[8].valid := 1, [67].log_data[9].min := 1.0, [67].log_data[9].max := 1.0, [67].log_data[9].total := 3599.5, [67].log_data[9].time := 3599.5, [67].log_data[9].valid := 1, [67].log_data[10].min := 1.0, [67].log_data[10].max := 1.0, [67].log_data[10].total := 3599.5, [67].log_data[10].time := 3599.5, [67].log_data[10].valid := 1, [67].log_data[11].time := 3599.5, [67].log_data[11].valid := 1, [67].log_data[12].min := 1.0, [67].log_data[12].max := 1.0, [67].log_data[12].total := 3599.5, [67].log_data[12].time := 3599.5, [67].log_data[12].valid := 1, [67].log_data[13].min := 1.0, [67].log_data[13].max := 1.0, [67].log_data[13].total := 3599.5, [67].log_data[13].time := 3599.5, [67].log_data[13].valid := 1, [67].log_data[14].time := 3599.5, [67].log_data[14].valid := 1, [67].log_data[15].time := 3599.5, [67].log_data[15].valid := 1, [67].log_data[16].time := 3599.5, [67].log_data[16].valid := 1, [67].log_data[17].min := 1.0, [67].log_data[17].max := 1.0, [67].log_data[17].total := 3599.5,
        [67].log_data[17].time := 3599.5, [67].log_data[17].valid := 1, [67].log_data[18].time := 3599.5, [67].log_data[18].valid := 1, [67].log_data[19].time := 3599.5, [67].log_data[19].valid := 1, [67].log_data[20].time := 3599.5, [67].log_data[20].valid := 1, [67].log_data[21].min := 1.0, [67].log_data[21].max := 1.0, [67].log_data[21].total := 3599.5, [67].log_data[21].time := 3599.5, [67].log_data[21].valid := 1, [67].log_data[22].time := 3599.5, [67].log_data[22].valid := 1, [67].log_data[23].time := 3599.5, [67].log_data[23].valid := 1, [67].log_data[24].time := 3599.5, [67].log_data[24].valid := 1, [67].log_data[25].time := 3599.5, [67].log_data[25].valid := 1, [67].log_data[26].time := 3599.5, [67].log_data[26].valid := 1, [67].log_data[27].time := 3599.5, [67].log_data[27].valid := 1, [67].log_data[28].time := 3599.5, [67].log_data[28].valid := 1, [67].log_data[29].min := 1.0, [67].log_data[29].max := 1.0, [67].log_data[29].total := 3599.5, [67].log_data[29].time := 3599.5, [67].log_data[29].valid := 1, [67].log_data[30].min := 1.0, [67].log_data[30].max := 1.0, [67].log_data[30].total := 3599.5, [67].log_data[30].time := 3599.5, [67].log_data[30].valid := 1, [67].log_data[31].max := 1.0, [67].log_data[31].total := 1626.998, [67].log_data[31].time := 3599.5, [67].log_data[31].minminute := 9, [67].log_data[31].valid := 1, [67].log_data[32].max := 1.0, [67].log_data[32].total := 1531.2471, [67].log_data[32].time := 3599.5, [67].log_data[32].maxminute := 10, [67].log_data[32].valid := 1, [67].log_data[33].time := 3599.5, [67].log_data[33].valid := 1, [67].log_data[34].time := 3599.5, [67].log_data[34].valid := 1, [67].log_data[35].max := 1.0, [67].log_data[35].total := 1629.7471, [67].log_data[35].time := 3599.5, [67].log_data[35].maxminute := 4, [67].log_data[35].valid := 1, [67].log_data[36].max := 1.0, [67].log_data[36].total := 1440.498, [67].log_data[36].time := 3599.5, [67].log_data[36].minminute := 2,
        [67].log_data[36].valid := 1, [67].log_data[37].max := 7.578351, [67].log_data[37].total := 3561.7556, [67].log_data[37].time := 3599.5, [67].log_data[37].maxminute := 43, [67].log_data[37].valid := 1, [67].log_data[38].time := 3599.5, [67].log_data[38].valid := 1, [67].log_data[39].min := 0.9981217, [67].log_data[39].max := 1.0213233, [67].log_data[39].total := 3624.951, [67].log_data[39].time := 3599.5, [67].log_data[39].minminute := 50, [67].log_data[39].maxminute := 44, [67].log_data[39].valid := 1, [67].log_data[40].min := 7.587675, [67].log_data[40].max := 7.597843, [67].log_data[40].total := 27327.514, [67].log_data[40].time := 3599.5, [67].log_data[40].minminute := 11, [67].log_data[40].maxminute := 15, [67].log_data[40].valid := 1, [67].log_data[41].min := 0.023717772, [67].log_data[41].max := 0.04138403, [67].log_data[41].total := 128.2696, [67].log_data[41].time := 3599.5, [67].log_data[41].minminute := 3, [67].log_data[41].maxminute := 20, [67].log_data[41].valid := 1, [67].log_data[42].min := 2.291525, [67].log_data[42].max := 2.2968247, [67].log_data[42].total := 8258.887, [67].log_data[42].time := 3599.5, [67].log_data[42].minminute := 58, [67].log_data[42].maxminute := 50, [67].log_data[42].valid := 1, [67].log_data[43].min := -0.27999878, [67].log_data[43].max := -0.26000214, [67].log_data[43].total := -976.3203, [67].log_data[43].time := 3599.5, [67].log_data[43].valid := 1, [67].log_data[44].min := -0.30000305, [67].log_data[44].max := -0.30000305, [67].log_data[44].total := -1079.941, [67].log_data[44].time := 3599.5, [67].log_data[44].valid := 1, [67].log_data[45].time := 3599.5, [67].log_data[45].valid := 1, [67].log_data[46].time := 3599.5, [67].log_data[46].valid := 1, [67].log_data[47].time := 3599.5, [67].log_data[47].valid := 1, [67].log_data[48].min := 6.62255, [67].log_data[48].max := 6.975128, [67].log_data[48].total := 24368.453, [67].log_data[48].time := 3599.5, [67].log_data[48].maxminute := 45, [67].log_data[48].valid := 1, [67].log_data[49].min := 7.4914274, [67].log_data[49].max := 9.749563,
        [67].log_data[49].total := 32603.605, [67].log_data[49].time := 3599.5, [67].log_data[49].minminute := 59, [67].log_data[49].maxminute := 42, [67].log_data[49].valid := 1, [67].log_data[50].min := 2.1958919, [67].log_data[50].max := 2.3037734, [67].log_data[50].total := 8070.347, [67].log_data[50].time := 3599.5, [67].log_data[50].minminute := 44, [67].log_data[50].maxminute := 52, [67].log_data[50].valid := 1, [67].log_data[51].time := 3599.5, [67].log_data[51].valid := 1, [67].log_data[52].min := -3.0200043, [67].log_data[52].max := 0.11999512, [67].log_data[52].total := -8017.77, [67].log_data[52].time := 3599.5, [67].log_data[52].maxminute := 9, [67].log_data[52].valid := 1, [67].log_data[53].min := -2.5800018, [67].log_data[53].max := 0.22000122, [67].log_data[53].total := -7290.7974, [67].log_data[53].time := 3599.5, [67].log_data[53].minminute := 48, [67].log_data[53].maxminute := 4, [67].log_data[53].valid := 1, [67].log_data[54].max := 0.554, [67].log_data[54].total := 1253.2957, [67].log_data[54].time := 3599.5, [67].log_data[54].maxminute := 42, [67].log_data[54].valid := 1, [67].log_data[55].max := 0.52099997, [67].log_data[55].total := 1217.2324, [67].log_data[55].time := 3599.5, [67].log_data[55].minminute := 2, [67].log_data[55].maxminute := 25, [67].log_data[55].valid := 1, [67].log_data[56].min := 0.16008857, [67].log_data[56].max := 0.1605204, [67].log_data[56].total := 576.85876, [67].log_data[56].time := 3599.5, [67].log_data[56].minminute := 1, [67].log_data[56].maxminute := 10, [67].log_data[56].valid := 1, [67].log_data[57].min := 0.26047197, [67].log_data[57].max := 0.2613357, [67].log_data[57].total := 938.1522, [67].log_data[57].time := 3599.5, [67].log_data[57].minminute := 3, [67].log_data[57].valid := 1, [67].log_data[58].time := 3599.5, [67].log_data[58].valid := 1, [67].log_data[59].time := 3599.5, [67].log_data[59].valid := 1, [67].log_data[60].valid := 1, [67].log_data[61].valid := 1, [67].log_data[62].valid := 1, [67].log_data[63].valid := 1, [67].log_data[64].valid := 1,
        [67].log_data[65].valid := 1, [67].log_data[66].valid := 1, [67].log_data[67].valid := 1, [67].log_data[68].valid := 1, [67].log_data[69].valid := 1, [67].log_data[70].valid := 1, [67].log_data[71].valid := 1, [67].log_data[72].valid := 1, [67].log_data[73].valid := 1, [67].log_data[74].valid := 1, [67].log_data[75].valid := 1, [67].log_data[76].valid := 1, [67].log_data[77].valid := 1, [67].log_data[78].valid := 1, [67].log_data[79].valid := 1, [67].log_data[80].valid := 1, [67].log_data[81].valid := 1, [67].log_data[82].valid := 1, [67].log_data[83].valid := 1, [67].log_data[84].valid := 1, [67].log_data[85].valid := 1, [67].log_data[86].valid := 1, [67].log_data[87].valid := 1, [67].log_data[88].valid := 1, [67].log_data[89].valid := 1, [67].log_data[90].valid := 1, [67].log_data[91].valid := 1, [67].log_data[92].valid := 1, [67].log_data[93].valid := 1, [67].log_data[94].valid := 1, [67].log_data[95].valid := 1, [67].log_data[96].valid := 1, [67].log_data[97].valid := 1, [67].log_data[98].valid := 1, [67].log_data[99].valid := 1, [67].log_data[100].valid := 1, [67].log_data[101].valid := 1, [67].log_data[102].valid := 1, [67].log_data[103].valid := 1, [67].log_data[104].valid := 1, [67].log_data[105].valid := 1, [67].log_data[106].valid := 1, [67].log_data[107].valid := 1, [67].log_data[108].valid := 1, [67].log_data[109].valid := 1, [67].log_data[110].valid := 1, [67].log_data[111].valid := 1, [67].log_data[112].valid := 1, [67].log_data[113].valid := 1, [67].log_data[114].valid := 1, [67].log_data[115].valid := 1, [67].log_data[116].valid := 1, [67].log_data[117].valid := 1, [67].log_data[118].valid := 1, [67].log_data[119].valid := 1, [67].log_data[120].valid := 1, [67].log_data[121].valid := 1, [67].log_data[122].valid := 1, [67].log_data[123].valid := 1, [67].log_data[124].valid := 1,
        [67].time.Year := 2023, [67].time.Month := 1, [67].time.Day := 15, [67].time.Hour := 22, [67].time.Minute := 59, [67].time.Second := 59, [68].log_data[0].min := 1.0, [68].log_data[0].max := 1.0, [68].log_data[0].total := 3600.0, [68].log_data[0].time := 3600.0, [68].log_data[0].valid := 1, [68].log_data[1].time := 3600.0, [68].log_data[1].valid := 1, [68].log_data[2].time := 3600.0, [68].log_data[2].valid := 1, [68].log_data[3].time := 3600.0, [68].log_data[3].valid := 1, [68].log_data[4].time := 3600.0, [68].log_data[4].valid := 1, [68].log_data[5].time := 3600.0, [68].log_data[5].valid := 1, [68].log_data[6].time := 3600.0, [68].log_data[6].valid := 1, [68].log_data[7].time := 3600.0, [68].log_data[7].valid := 1, [68].log_data[8].min := 1.0, [68].log_data[8].max := 1.0, [68].log_data[8].total := 3600.0, [68].log_data[8].time := 3600.0, [68].log_data[8].valid := 1, [68].log_data[9].min := 1.0, [68].log_data[9].max := 1.0, [68].log_data[9].total := 3600.0, [68].log_data[9].time := 3600.0, [68].log_data[9].valid := 1, [68].log_data[10].min := 1.0, [68].log_data[10].max := 1.0, [68].log_data[10].total := 3600.0, [68].log_data[10].time := 3600.0, [68].log_data[10].valid := 1, [68].log_data[11].time := 3600.0, [68].log_data[11].valid := 1, [68].log_data[12].min := 1.0, [68].log_data[12].max := 1.0, [68].log_data[12].total := 3600.0, [68].log_data[12].time := 3600.0, [68].log_data[12].valid := 1, [68].log_data[13].min := 1.0, [68].log_data[13].max := 1.0, [68].log_data[13].total := 3600.0, [68].log_data[13].time := 3600.0, [68].log_data[13].valid := 1, [68].log_data[14].time := 3600.0, [68].log_data[14].valid := 1, [68].log_data[15].time := 3600.0, [68].log_data[15].valid := 1, [68].log_data[16].time := 3600.0, [68].log_data[16].valid := 1, [68].log_data[17].min := 1.0, [68].log_data[17].max := 1.0,
        [68].log_data[17].total := 3600.0, [68].log_data[17].time := 3600.0, [68].log_data[17].valid := 1, [68].log_data[18].time := 3600.0, [68].log_data[18].valid := 1, [68].log_data[19].time := 3600.0, [68].log_data[19].valid := 1, [68].log_data[20].time := 3600.0, [68].log_data[20].valid := 1, [68].log_data[21].min := 1.0, [68].log_data[21].max := 1.0, [68].log_data[21].total := 3600.0, [68].log_data[21].time := 3600.0, [68].log_data[21].valid := 1, [68].log_data[22].time := 3600.0, [68].log_data[22].valid := 1, [68].log_data[23].time := 3600.0, [68].log_data[23].valid := 1, [68].log_data[24].time := 3600.0, [68].log_data[24].valid := 1, [68].log_data[25].time := 3600.0, [68].log_data[25].valid := 1, [68].log_data[26].time := 3600.0, [68].log_data[26].valid := 1, [68].log_data[27].time := 3600.0, [68].log_data[27].valid := 1, [68].log_data[28].time := 3600.0, [68].log_data[28].valid := 1, [68].log_data[29].min := 1.0, [68].log_data[29].max := 1.0, [68].log_data[29].total := 3600.0, [68].log_data[29].time := 3600.0, [68].log_data[29].valid := 1, [68].log_data[30].min := 1.0, [68].log_data[30].max := 1.0, [68].log_data[30].total := 3600.0, [68].log_data[30].time := 3600.0, [68].log_data[30].valid := 1, [68].log_data[31].max := 1.0, [68].log_data[31].total := 1629.7471, [68].log_data[31].time := 3600.0, [68].log_data[31].maxminute := 3, [68].log_data[31].valid := 1, [68].log_data[32].max := 1.0, [68].log_data[32].total := 1441.249, [68].log_data[32].time := 3600.0, [68].log_data[32].minminute := 1, [68].log_data[32].valid := 1, [68].log_data[33].time := 3600.0, [68].log_data[33].valid := 1, [68].log_data[34].time := 3600.0, [68].log_data[34].valid := 1, [68].log_data[35].max := 1.0, [68].log_data[35].total := 1629.7471, [68].log_data[35].time := 3600.0, [68].log_data[35].maxminute := 7, [68].log_data[35].valid := 1, [68].log_data[36].max := 1.0, [68].log_data[36].total := 1440.498, [68].log_data[36].time := 3600.0,
        [68].log_data[36].minminute := 5, [68].log_data[36].valid := 1, [68].log_data[37].time := 3600.0, [68].log_data[37].valid := 1, [68].log_data[38].time := 3600.0, [68].log_data[38].valid := 1, [68].log_data[39].min := 0.9992994, [68].log_data[39].max := 1.0100169, [68].log_data[39].total := 3620.4727, [68].log_data[39].time := 3600.0, [68].log_data[39].minminute := 8, [68].log_data[39].maxminute := 48, [68].log_data[39].valid := 1, [68].log_data[40].min := 7.574485, [68].log_data[40].max := 7.597843, [68].log_data[40].total := 27321.938, [68].log_data[40].time := 3600.0, [68].log_data[40].minminute := 52, [68].log_data[40].maxminute := 48, [68].log_data[40].valid := 1, [68].log_data[41].min := 0.022540038, [68].log_data[41].max := 0.03215845, [68].log_data[41].total := 92.32604, [68].log_data[41].time := 3600.0, [68].log_data[41].minminute := 16, [68].log_data[41].maxminute := 21, [68].log_data[41].valid := 1, [68].log_data[42].min := 2.291407, [68].log_data[42].max := 2.2964714, [68].log_data[42].total := 8259.999, [68].log_data[42].time := 3600.0, [68].log_data[42].minminute := 16, [68].log_data[42].maxminute := 1, [68].log_data[42].valid := 1, [68].log_data[43].min := -0.27999878, [68].log_data[43].max := -0.26000214, [68].log_data[43].total := -973.92584, [68].log_data[43].time := 3600.0, [68].log_data[43].valid := 1, [68].log_data[44].min := -0.3199997, [68].log_data[44].max := -0.30000305, [68].log_data[44].total := -1080.0962, [68].log_data[44].time := 3600.0, [68].log_data[44].minminute := 14, [68].log_data[44].valid := 1, [68].log_data[45].time := 3600.0, [68].log_data[45].valid := 1, [68].log_data[46].time := 3600.0, [68].log_data[46].valid := 1, [68].log_data[47].time := 3600.0, [68].log_data[47].valid := 1, [68].log_data[48].min := 6.5807796, [68].log_data[48].max := 6.7912817, [68].log_data[48].total := 24180.096, [68].log_data[48].time := 3600.0, [68].log_data[48].minminute := 17, [68].log_data[48].maxminute := 31, [68].log_data[48].valid := 1, [68].log_data[49].min := 7.0841227, [68].log_data[49].max := 9.741712,
        [68].log_data[49].total := 30669.473, [68].log_data[49].time := 3600.0, [68].log_data[49].minminute := 9, [68].log_data[49].maxminute := 59, [68].log_data[49].valid := 1, [68].log_data[50].min := 2.2139113, [68].log_data[50].max := 2.297296, [68].log_data[50].total := 8128.645, [68].log_data[50].time := 3600.0, [68].log_data[50].minminute := 59, [68].log_data[50].valid := 1, [68].log_data[51].time := 3600.0, [68].log_data[51].valid := 1, [68].log_data[52].min := -3.0800018, [68].log_data[52].max := 0.11999512, [68].log_data[52].total := -7793.837, [68].log_data[52].time := 3600.0, [68].log_data[52].minminute := 45, [68].log_data[52].maxminute := 1, [68].log_data[52].valid := 1, [68].log_data[53].min := -2.600006, [68].log_data[53].max := 0.22000122, [68].log_data[53].total := -7306.6826, [68].log_data[53].time := 3600.0, [68].log_data[53].minminute := 57, [68].log_data[53].maxminute := 17, [68].log_data[53].valid := 1, [68].log_data[54].max := 0.5525, [68].log_data[54].total := 1217.4211, [68].log_data[54].time := 3600.0, [68].log_data[54].minminute := 1, [68].log_data[54].maxminute := 45, [68].log_data[54].valid := 1, [68].log_data[55].max := 0.5145, [68].log_data[55].total := 1217.4083, [68].log_data[55].time := 3600.0, [68].log_data[55].minminute := 5, [68].log_data[55].maxminute := 7, [68].log_data[55].valid := 1, [68].log_data[56].min := 0.16001005, [68].log_data[56].max := 0.16048115, [68].log_data[56].total := 576.82935, [68].log_data[56].time := 3600.0, [68].log_data[56].minminute := 14, [68].log_data[56].maxminute := 46, [68].log_data[56].valid := 1, [68].log_data[57].min := 0.25890166, [68].log_data[57].max := 0.2608646, [68].log_data[57].total := 934.3687, [68].log_data[57].time := 3600.0, [68].log_data[57].minminute := 33, [68].log_data[57].maxminute := 4, [68].log_data[57].valid := 1, [68].log_data[58].time := 3600.0, [68].log_data[58].valid := 1, [68].log_data[59].time := 3600.0, [68].log_data[59].valid := 1, [68].log_data[60].valid := 1, [68].log_data[61].valid := 1, [68].log_data[62].valid := 1,
        [68].log_data[63].valid := 1, [68].log_data[64].valid := 1, [68].log_data[65].valid := 1, [68].log_data[66].valid := 1, [68].log_data[67].valid := 1, [68].log_data[68].valid := 1, [68].log_data[69].valid := 1, [68].log_data[70].valid := 1, [68].log_data[71].valid := 1, [68].log_data[72].valid := 1, [68].log_data[73].valid := 1, [68].log_data[74].valid := 1, [68].log_data[75].valid := 1, [68].log_data[76].valid := 1, [68].log_data[77].valid := 1, [68].log_data[78].valid := 1, [68].log_data[79].valid := 1, [68].log_data[80].valid := 1, [68].log_data[81].valid := 1, [68].log_data[82].valid := 1, [68].log_data[83].valid := 1, [68].log_data[84].valid := 1, [68].log_data[85].valid := 1, [68].log_data[86].valid := 1, [68].log_data[87].valid := 1, [68].log_data[88].valid := 1, [68].log_data[89].valid := 1, [68].log_data[90].valid := 1, [68].log_data[91].valid := 1, [68].log_data[92].valid := 1, [68].log_data[93].valid := 1, [68].log_data[94].valid := 1, [68].log_data[95].valid := 1, [68].log_data[96].valid := 1, [68].log_data[97].valid := 1, [68].log_data[98].valid := 1, [68].log_data[99].valid := 1, [68].log_data[100].valid := 1, [68].log_data[101].valid := 1, [68].log_data[102].valid := 1, [68].log_data[103].valid := 1, [68].log_data[104].valid := 1, [68].log_data[105].valid := 1, [68].log_data[106].valid := 1, [68].log_data[107].valid := 1, [68].log_data[108].valid := 1, [68].log_data[109].valid := 1, [68].log_data[110].valid := 1, [68].log_data[111].valid := 1, [68].log_data[112].valid := 1, [68].log_data[113].valid := 1, [68].log_data[114].valid := 1, [68].log_data[115].valid := 1, [68].log_data[116].valid := 1, [68].log_data[117].valid := 1, [68].log_data[118].valid := 1, [68].log_data[119].valid := 1, [68].log_data[120].valid := 1, [68].log_data[121].valid := 1, [68].log_data[122].valid := 1,
        [68].log_data[123].valid := 1, [68].log_data[124].valid := 1, [68].time.Year := 2023, [68].time.Month := 1, [68].time.Day := 15, [68].time.Hour := 23, [68].time.Minute := 59, [68].time.Second := 59, [69].log_data[0].min := 1.0, [69].log_data[0].max := 1.0, [69].log_data[0].total := 3600.0, [69].log_data[0].time := 3600.0, [69].log_data[0].valid := 1, [69].log_data[1].max := 1.0, [69].log_data[1].total := 547.0, [69].log_data[1].time := 3600.0, [69].log_data[1].maxminute := 14, [69].log_data[1].valid := 1, [69].log_data[2].max := 1.0, [69].log_data[2].total := 543.5, [69].log_data[2].time := 3600.0, [69].log_data[2].maxminute := 14, [69].log_data[2].valid := 1, [69].log_data[3].time := 3600.0, [69].log_data[3].valid := 1, [69].log_data[4].time := 3600.0, [69].log_data[4].valid := 1, [69].log_data[5].max := 1.0, [69].log_data[5].total := 249.5, [69].log_data[5].time := 3600.0, [69].log_data[5].maxminute := 16, [69].log_data[5].valid := 1, [69].log_data[6].time := 3600.0, [69].log_data[6].valid := 1, [69].log_data[7].time := 3600.0, [69].log_data[7].valid := 1, [69].log_data[8].min := 1.0, [69].log_data[8].max := 1.0, [69].log_data[8].total := 3600.0, [69].log_data[8].time := 3600.0, [69].log_data[8].valid := 1, [69].log_data[9].min := 1.0, [69].log_data[9].max := 1.0, [69].log_data[9].total := 3600.0, [69].log_data[9].time := 3600.0, [69].log_data[9].valid := 1, [69].log_data[10].min := 1.0, [69].log_data[10].max := 1.0, [69].log_data[10].total := 3600.0, [69].log_data[10].time := 3600.0, [69].log_data[10].valid := 1, [69].log_data[11].time := 3600.0, [69].log_data[11].valid := 1, [69].log_data[12].min := 1.0, [69].log_data[12].max := 1.0, [69].log_data[12].total := 3600.0, [69].log_data[12].time := 3600.0, [69].log_data[12].valid := 1, [69].log_data[13].min := 1.0, [69].log_data[13].max := 1.0,
        [69].log_data[13].total := 3600.0, [69].log_data[13].time := 3600.0, [69].log_data[13].valid := 1, [69].log_data[14].time := 3600.0, [69].log_data[14].valid := 1, [69].log_data[15].time := 3600.0, [69].log_data[15].valid := 1, [69].log_data[16].time := 3600.0, [69].log_data[16].valid := 1, [69].log_data[17].min := 1.0, [69].log_data[17].max := 1.0, [69].log_data[17].total := 3600.0, [69].log_data[17].time := 3600.0, [69].log_data[17].valid := 1, [69].log_data[18].time := 3600.0, [69].log_data[18].valid := 1, [69].log_data[19].time := 3600.0, [69].log_data[19].valid := 1, [69].log_data[20].time := 3600.0, [69].log_data[20].valid := 1, [69].log_data[21].min := 1.0, [69].log_data[21].max := 1.0, [69].log_data[21].total := 3600.0, [69].log_data[21].time := 3600.0, [69].log_data[21].valid := 1, [69].log_data[22].time := 3600.0, [69].log_data[22].valid := 1, [69].log_data[23].time := 3600.0, [69].log_data[23].valid := 1, [69].log_data[24].time := 3600.0, [69].log_data[24].valid := 1, [69].log_data[25].time := 3600.0, [69].log_data[25].valid := 1, [69].log_data[26].time := 3600.0, [69].log_data[26].valid := 1, [69].log_data[27].time := 3600.0, [69].log_data[27].valid := 1, [69].log_data[28].time := 3600.0, [69].log_data[28].valid := 1, [69].log_data[29].min := 1.0, [69].log_data[29].max := 1.0, [69].log_data[29].total := 3600.0, [69].log_data[29].time := 3600.0, [69].log_data[29].valid := 1, [69].log_data[30].min := 1.0, [69].log_data[30].max := 1.0, [69].log_data[30].total := 3600.0, [69].log_data[30].time := 3600.0, [69].log_data[30].valid := 1, [69].log_data[31].max := 1.0, [69].log_data[31].total := 1629.998, [69].log_data[31].time := 3600.0, [69].log_data[31].maxminute := 6, [69].log_data[31].valid := 1, [69].log_data[32].max := 1.0, [69].log_data[32].total := 1440.998, [69].log_data[32].time := 3600.0, [69].log_data[32].minminute := 4, [69].log_data[32].valid := 1, [69].log_data[33].time := 3600.0,
        [69].log_data[33].valid := 1, [69].log_data[34].time := 3600.0, [69].log_data[34].valid := 1, [69].log_data[35].max := 1.0, [69].log_data[35].total := 1540.7471, [69].log_data[35].time := 3600.0, [69].log_data[35].maxminute := 10, [69].log_data[35].valid := 1, [69].log_data[36].max := 1.0, [69].log_data[36].total := 1617.998, [69].log_data[36].time := 3600.0, [69].log_data[36].minminute := 8, [69].log_data[36].valid := 1, [69].log_data[37].max := 7.3333793, [69].log_data[37].total := 3484.0579, [69].log_data[37].time := 3600.0, [69].log_data[37].maxminute := 16, [69].log_data[37].valid := 1, [69].log_data[38].time := 3600.0, [69].log_data[38].valid := 1, [69].log_data[39].min := 0.99376404, [69].log_data[39].max := 1.0219122, [69].log_data[39].total := 3613.488, [69].log_data[39].time := 3600.0, [69].log_data[39].minminute := 35, [69].log_data[39].maxminute := 21, [69].log_data[39].valid := 1, [69].log_data[40].min := 7.577233, [69].log_data[40].max := 7.609111, [69].log_data[40].total := 27325.998, [69].log_data[40].time := 3600.0, [69].log_data[40].minminute := 43, [69].log_data[40].maxminute := 51, [69].log_data[40].valid := 1, [69].log_data[41].min := 0.022540038, [69].log_data[41].max := 0.0384397, [69].log_data[41].total := 93.73055, [69].log_data[41].time := 3600.0, [69].log_data[41].minminute := 41, [69].log_data[41].maxminute := 15, [69].log_data[41].valid := 1, [69].log_data[42].min := 2.2917604, [69].log_data[42].max := 2.2965894, [69].log_data[42].total := 8259.81, [69].log_data[42].time := 3600.0, [69].log_data[42].minminute := 29, [69].log_data[42].valid := 1, [69].log_data[43].min := -0.27999878, [69].log_data[43].max := -0.26000214, [69].log_data[43].total := -966.9633, [69].log_data[43].time := 3600.0, [69].log_data[43].valid := 1, [69].log_data[44].min := -0.30000305, [69].log_data[44].max := -0.30000305, [69].log_data[44].total := -1080.0911, [69].log_data[44].time := 3600.0, [69].log_data[44].valid := 1, [69].log_data[45].time := 3600.0, [69].log_data[45].valid := 1, [69].log_data[46].time := 3600.0,
        [69].log_data[46].valid := 1, [69].log_data[47].time := 3600.0, [69].log_data[47].valid := 1, [69].log_data[48].min := 6.583802, [69].log_data[48].max := 6.984747, [69].log_data[48].total := 24229.898, [69].log_data[48].time := 3600.0, [69].log_data[48].minminute := 48, [69].log_data[48].maxminute := 23, [69].log_data[48].valid := 1, [69].log_data[49].min := 7.0994334, [69].log_data[49].max := 9.791766, [69].log_data[49].total := 30162.012, [69].log_data[49].time := 3600.0, [69].log_data[49].minminute := 41, [69].log_data[49].maxminute := 12, [69].log_data[49].valid := 1, [69].log_data[50].min := 2.1912985, [69].log_data[50].max := 2.3016534, [69].log_data[50].total := 8126.911, [69].log_data[50].time := 3600.0, [69].log_data[50].minminute := 16, [69].log_data[50].maxminute := 23, [69].log_data[50].valid := 1, [69].log_data[51].time := 3600.0, [69].log_data[51].valid := 1, [69].log_data[52].min := -2.9800034, [69].log_data[52].max := 0.11999512, [69].log_data[52].total := -7832.6147, [69].log_data[52].time := 3600.0, [69].log_data[52].minminute := 6, [69].log_data[52].maxminute := 4, [69].log_data[52].valid := 1, [69].log_data[53].min := -2.7000046, [69].log_data[53].max := 0.22000122, [69].log_data[53].total := -7533.547, [69].log_data[53].time := 3600.0, [69].log_data[53].minminute := 52, [69].log_data[53].maxminute := 10, [69].log_data[53].valid := 1, [69].log_data[54].max := 0.55050004, [69].log_data[54].total := 1217.8053, [69].log_data[54].time := 3600.0, [69].log_data[54].minminute := 4, [69].log_data[54].maxminute := 48, [69].log_data[54].valid := 1, [69].log_data[55].max := 0.55550003, [69].log_data[55].total := 1253.638, [69].log_data[55].time := 3600.0, [69].log_data[55].minminute := 8, [69].log_data[55].maxminute := 52, [69].log_data[55].valid := 1, [69].log_data[56].min := 0.16001005, [69].log_data[56].max := 0.1605204, [69].log_data[56].total := 576.8503, [69].log_data[56].time := 3600.0, [69].log_data[56].minminute := 27, [69].log_data[56].maxminute := 30, [69].log_data[56].valid := 1, [69].log_data[57].min := 0.2573706,
        [69].log_data[57].max := 0.25929424, [69].log_data[57].total := 931.8406, [69].log_data[57].time := 3600.0, [69].log_data[57].minminute := 58, [69].log_data[57].maxminute := 32, [69].log_data[57].valid := 1, [69].log_data[58].time := 3600.0, [69].log_data[58].valid := 1, [69].log_data[59].time := 3600.0, [69].log_data[59].valid := 1, [69].log_data[60].valid := 1, [69].log_data[61].valid := 1, [69].log_data[62].valid := 1, [69].log_data[63].valid := 1, [69].log_data[64].valid := 1, [69].log_data[65].valid := 1, [69].log_data[66].valid := 1, [69].log_data[67].valid := 1, [69].log_data[68].valid := 1, [69].log_data[69].valid := 1, [69].log_data[70].valid := 1, [69].log_data[71].valid := 1, [69].log_data[72].valid := 1, [69].log_data[73].valid := 1, [69].log_data[74].valid := 1, [69].log_data[75].valid := 1, [69].log_data[76].valid := 1, [69].log_data[77].valid := 1, [69].log_data[78].valid := 1, [69].log_data[79].valid := 1, [69].log_data[80].valid := 1, [69].log_data[81].valid := 1, [69].log_data[82].valid := 1, [69].log_data[83].valid := 1, [69].log_data[84].valid := 1, [69].log_data[85].valid := 1, [69].log_data[86].valid := 1, [69].log_data[87].valid := 1, [69].log_data[88].valid := 1, [69].log_data[89].valid := 1, [69].log_data[90].valid := 1, [69].log_data[91].valid := 1, [69].log_data[92].valid := 1, [69].log_data[93].valid := 1, [69].log_data[94].valid := 1, [69].log_data[95].valid := 1, [69].log_data[96].valid := 1, [69].log_data[97].valid := 1, [69].log_data[98].valid := 1, [69].log_data[99].valid := 1, [69].log_data[100].valid := 1, [69].log_data[101].valid := 1, [69].log_data[102].valid := 1, [69].log_data[103].valid := 1, [69].log_data[104].valid := 1, [69].log_data[105].valid := 1, [69].log_data[106].valid := 1, [69].log_data[107].valid := 1, [69].log_data[108].valid := 1, [69].log_data[109].valid := 1,
        [69].log_data[110].valid := 1, [69].log_data[111].valid := 1, [69].log_data[112].valid := 1, [69].log_data[113].valid := 1, [69].log_data[114].valid := 1, [69].log_data[115].valid := 1, [69].log_data[116].valid := 1, [69].log_data[117].valid := 1, [69].log_data[118].valid := 1, [69].log_data[119].valid := 1, [69].log_data[120].valid := 1, [69].log_data[121].valid := 1, [69].log_data[122].valid := 1, [69].log_data[123].valid := 1, [69].log_data[124].valid := 1, [69].time.Year := 2023, [69].time.Month := 1, [69].time.Day := 16, [69].time.Minute := 59, [69].time.Second := 59, [70].log_data[0].min := 1.0, [70].log_data[0].max := 1.0, [70].log_data[0].total := 3600.0, [70].log_data[0].time := 3600.0, [70].log_data[0].valid := 1, [70].log_data[1].time := 3600.0, [70].log_data[1].valid := 1, [70].log_data[2].time := 3600.0, [70].log_data[2].valid := 1, [70].log_data[3].time := 3600.0, [70].log_data[3].valid := 1, [70].log_data[4].time := 3600.0, [70].log_data[4].valid := 1, [70].log_data[5].time := 3600.0, [70].log_data[5].valid := 1, [70].log_data[6].time := 3600.0, [70].log_data[6].valid := 1, [70].log_data[7].time := 3600.0, [70].log_data[7].valid := 1, [70].log_data[8].min := 1.0, [70].log_data[8].max := 1.0, [70].log_data[8].total := 3600.0, [70].log_data[8].time := 3600.0, [70].log_data[8].valid := 1, [70].log_data[9].min := 1.0, [70].log_data[9].max := 1.0, [70].log_data[9].total := 3600.0, [70].log_data[9].time := 3600.0, [70].log_data[9].valid := 1, [70].log_data[10].min := 1.0, [70].log_data[10].max := 1.0, [70].log_data[10].total := 3600.0, [70].log_data[10].time := 3600.0, [70].log_data[10].valid := 1, [70].log_data[11].time := 3600.0, [70].log_data[11].valid := 1, [70].log_data[12].min := 1.0, [70].log_data[12].max := 1.0, [70].log_data[12].total := 3600.0, [70].log_data[12].time := 3600.0,
        [70].log_data[12].valid := 1, [70].log_data[13].min := 1.0, [70].log_data[13].max := 1.0, [70].log_data[13].total := 3600.0, [70].log_data[13].time := 3600.0, [70].log_data[13].valid := 1, [70].log_data[14].time := 3600.0, [70].log_data[14].valid := 1, [70].log_data[15].time := 3600.0, [70].log_data[15].valid := 1, [70].log_data[16].time := 3600.0, [70].log_data[16].valid := 1, [70].log_data[17].min := 1.0, [70].log_data[17].max := 1.0, [70].log_data[17].total := 3600.0, [70].log_data[17].time := 3600.0, [70].log_data[17].valid := 1, [70].log_data[18].time := 3600.0, [70].log_data[18].valid := 1, [70].log_data[19].time := 3600.0, [70].log_data[19].valid := 1, [70].log_data[20].time := 3600.0, [70].log_data[20].valid := 1, [70].log_data[21].min := 1.0, [70].log_data[21].max := 1.0, [70].log_data[21].total := 3600.0, [70].log_data[21].time := 3600.0, [70].log_data[21].valid := 1, [70].log_data[22].time := 3600.0, [70].log_data[22].valid := 1, [70].log_data[23].time := 3600.0, [70].log_data[23].valid := 1, [70].log_data[24].time := 3600.0, [70].log_data[24].valid := 1, [70].log_data[25].time := 3600.0, [70].log_data[25].valid := 1, [70].log_data[26].time := 3600.0, [70].log_data[26].valid := 1, [70].log_data[27].time := 3600.0, [70].log_data[27].valid := 1, [70].log_data[28].time := 3600.0, [70].log_data[28].valid := 1, [70].log_data[29].min := 1.0, [70].log_data[29].max := 1.0, [70].log_data[29].total := 3600.0, [70].log_data[29].time := 3600.0, [70].log_data[29].valid := 1, [70].log_data[30].min := 1.0, [70].log_data[30].max := 1.0, [70].log_data[30].total := 3600.0, [70].log_data[30].time := 3600.0, [70].log_data[30].valid := 1, [70].log_data[31].max := 1.0, [70].log_data[31].total := 1595.7471, [70].log_data[31].time := 3600.0, [70].log_data[31].maxminute := 9, [70].log_data[31].valid := 1, [70].log_data[32].max := 1.0, [70].log_data[32].total := 1563.249, [70].log_data[32].time := 3600.0,
        [70].log_data[32].minminute := 7, [70].log_data[32].valid := 1, [70].log_data[33].time := 3600.0, [70].log_data[33].valid := 1, [70].log_data[34].time := 3600.0, [70].log_data[34].valid := 1, [70].log_data[35].max := 1.0, [70].log_data[35].total := 1440.7471, [70].log_data[35].time := 3600.0, [70].log_data[35].minminute := 1, [70].log_data[35].valid := 1, [70].log_data[36].max := 1.0, [70].log_data[36].total := 1629.7471, [70].log_data[36].time := 3600.0, [70].log_data[36].maxminute := 2, [70].log_data[36].valid := 1, [70].log_data[37].time := 3600.0, [70].log_data[37].valid := 1, [70].log_data[38].time := 3600.0, [70].log_data[38].valid := 1, [70].log_data[39].min := 0.99376404, [70].log_data[39].max := 1.0066015, [70].log_data[39].total := 3606.7202, [70].log_data[39].time := 3600.0, [70].log_data[39].minminute := 34, [70].log_data[39].maxminute := 12, [70].log_data[39].valid := 1, [70].log_data[40].min := 7.5571713, [70].log_data[40].max := 7.6121335, [70].log_data[40].total := 27330.541, [70].log_data[40].time := 3600.0, [70].log_data[40].minminute := 42, [70].log_data[40].maxminute := 46, [70].log_data[40].valid := 1, [70].log_data[41].min := 0.022540038, [70].log_data[41].max := 0.04432837, [70].log_data[41].total := 113.93812, [70].log_data[41].time := 3600.0, [70].log_data[41].minminute := 3, [70].log_data[41].maxminute := 31, [70].log_data[41].valid := 1, [70].log_data[42].min := 2.291525, [70].log_data[42].max := 2.2963536, [70].log_data[42].total := 8259.704, [70].log_data[42].time := 3600.0, [70].log_data[42].minminute := 9, [70].log_data[42].maxminute := 3, [70].log_data[42].valid := 1, [70].log_data[43].min := -0.27999878, [70].log_data[43].max := -0.26000214, [70].log_data[43].total := -994.549, [70].log_data[43].time := 3600.0, [70].log_data[43].valid := 1, [70].log_data[44].min := -0.30000305, [70].log_data[44].max := -0.30000305, [70].log_data[44].total := -1080.0911, [70].log_data[44].time := 3600.0, [70].log_data[44].valid := 1, [70].log_data[45].time := 3600.0, [70].log_data[45].valid := 1,
        [70].log_data[46].time := 3600.0, [70].log_data[46].valid := 1, [70].log_data[47].time := 3600.0, [70].log_data[47].valid := 1, [70].log_data[48].min := 6.742091, [70].log_data[48].max := 6.8096943, [70].log_data[48].total := 24414.893, [70].log_data[48].time := 3600.0, [70].log_data[48].maxminute := 6, [70].log_data[48].valid := 1, [70].log_data[49].min := 8.344117, [70].log_data[49].max := 9.782736, [70].log_data[49].total := 34273.527, [70].log_data[49].time := 3600.0, [70].log_data[49].maxminute := 42, [70].log_data[49].valid := 1, [70].log_data[50].min := 2.1753988, [70].log_data[50].max := 2.26373, [70].log_data[50].total := 7991.6616, [70].log_data[50].time := 3600.0, [70].log_data[50].minminute := 59, [70].log_data[50].valid := 1, [70].log_data[51].time := 3600.0, [70].log_data[51].valid := 1, [70].log_data[52].min := -2.9800034, [70].log_data[52].max := 0.11999512, [70].log_data[52].total := -8086.444, [70].log_data[52].time := 3600.0, [70].log_data[52].minminute := 51, [70].log_data[52].maxminute := 8, [70].log_data[52].valid := 1, [70].log_data[53].min := -2.600006, [70].log_data[53].max := 0.2599945, [70].log_data[53].total := -7354.7617, [70].log_data[53].time := 3600.0, [70].log_data[53].minminute := 57, [70].log_data[53].maxminute := 23, [70].log_data[53].valid := 1, [70].log_data[54].max := 0.538, [70].log_data[54].total := 1254.6964, [70].log_data[54].time := 3600.0, [70].log_data[54].minminute := 7, [70].log_data[54].maxminute := 30, [70].log_data[54].valid := 1, [70].log_data[55].max := 0.518, [70].log_data[55].total := 1217.0277, [70].log_data[55].time := 3600.0, [70].log_data[55].minminute := 1, [70].log_data[55].maxminute := 45, [70].log_data[55].valid := 1, [70].log_data[56].min := 0.16001005, [70].log_data[56].max := 0.1605204, [70].log_data[56].total := 576.941, [70].log_data[56].time := 3600.0, [70].log_data[56].minminute := 3, [70].log_data[56].maxminute := 3, [70].log_data[56].valid := 1, [70].log_data[57].min := 0.25733134, [70].log_data[57].max := 0.25776318, [70].log_data[57].total := 927.1579,
        [70].log_data[57].time := 3600.0, [70].log_data[57].minminute := 4, [70].log_data[57].maxminute := 9, [70].log_data[57].valid := 1, [70].log_data[58].time := 3600.0, [70].log_data[58].valid := 1, [70].log_data[59].time := 3600.0, [70].log_data[59].valid := 1, [70].log_data[60].valid := 1, [70].log_data[61].valid := 1, [70].log_data[62].valid := 1, [70].log_data[63].valid := 1, [70].log_data[64].valid := 1, [70].log_data[65].valid := 1, [70].log_data[66].valid := 1, [70].log_data[67].valid := 1, [70].log_data[68].valid := 1, [70].log_data[69].valid := 1, [70].log_data[70].valid := 1, [70].log_data[71].valid := 1, [70].log_data[72].valid := 1, [70].log_data[73].valid := 1, [70].log_data[74].valid := 1, [70].log_data[75].valid := 1, [70].log_data[76].valid := 1, [70].log_data[77].valid := 1, [70].log_data[78].valid := 1, [70].log_data[79].valid := 1, [70].log_data[80].valid := 1, [70].log_data[81].valid := 1, [70].log_data[82].valid := 1, [70].log_data[83].valid := 1, [70].log_data[84].valid := 1, [70].log_data[85].valid := 1, [70].log_data[86].valid := 1, [70].log_data[87].valid := 1, [70].log_data[88].valid := 1, [70].log_data[89].valid := 1, [70].log_data[90].valid := 1, [70].log_data[91].valid := 1, [70].log_data[92].valid := 1, [70].log_data[93].valid := 1, [70].log_data[94].valid := 1, [70].log_data[95].valid := 1, [70].log_data[96].valid := 1, [70].log_data[97].valid := 1, [70].log_data[98].valid := 1, [70].log_data[99].valid := 1, [70].log_data[100].valid := 1, [70].log_data[101].valid := 1, [70].log_data[102].valid := 1, [70].log_data[103].valid := 1, [70].log_data[104].valid := 1, [70].log_data[105].valid := 1, [70].log_data[106].valid := 1, [70].log_data[107].valid := 1, [70].log_data[108].valid := 1, [70].log_data[109].valid := 1, [70].log_data[110].valid := 1, [70].log_data[111].valid := 1,
        [70].log_data[112].valid := 1, [70].log_data[113].valid := 1, [70].log_data[114].valid := 1, [70].log_data[115].valid := 1, [70].log_data[116].valid := 1, [70].log_data[117].valid := 1, [70].log_data[118].valid := 1, [70].log_data[119].valid := 1, [70].log_data[120].valid := 1, [70].log_data[121].valid := 1, [70].log_data[122].valid := 1, [70].log_data[123].valid := 1, [70].log_data[124].valid := 1, [70].time.Year := 2023, [70].time.Month := 1, [70].time.Day := 16, [70].time.Hour := 1, [70].time.Minute := 59, [70].time.Second := 59, [71].log_data[0].min := 1.0, [71].log_data[0].max := 1.0, [71].log_data[0].total := 3600.0, [71].log_data[0].time := 3600.0, [71].log_data[0].valid := 1, [71].log_data[1].max := 1.0, [71].log_data[1].total := 521.0, [71].log_data[1].time := 3600.0, [71].log_data[1].maxminute := 45, [71].log_data[1].valid := 1, [71].log_data[2].max := 1.0, [71].log_data[2].total := 517.5, [71].log_data[2].time := 3600.0, [71].log_data[2].maxminute := 46, [71].log_data[2].valid := 1, [71].log_data[3].time := 3600.0, [71].log_data[3].valid := 1, [71].log_data[4].time := 3600.0, [71].log_data[4].valid := 1, [71].log_data[5].max := 1.0, [71].log_data[5].total := 229.5, [71].log_data[5].time := 3600.0, [71].log_data[5].maxminute := 48, [71].log_data[5].valid := 1, [71].log_data[6].time := 3600.0, [71].log_data[6].valid := 1, [71].log_data[7].time := 3600.0, [71].log_data[7].valid := 1, [71].log_data[8].min := 1.0, [71].log_data[8].max := 1.0, [71].log_data[8].total := 3600.0, [71].log_data[8].time := 3600.0, [71].log_data[8].valid := 1, [71].log_data[9].min := 1.0, [71].log_data[9].max := 1.0, [71].log_data[9].total := 3600.0, [71].log_data[9].time := 3600.0, [71].log_data[9].valid := 1, [71].log_data[10].min := 1.0, [71].log_data[10].max := 1.0, [71].log_data[10].total := 3600.0,
        [71].log_data[10].time := 3600.0, [71].log_data[10].valid := 1, [71].log_data[11].time := 3600.0, [71].log_data[11].valid := 1, [71].log_data[12].min := 1.0, [71].log_data[12].max := 1.0, [71].log_data[12].total := 3600.0, [71].log_data[12].time := 3600.0, [71].log_data[12].valid := 1, [71].log_data[13].min := 1.0, [71].log_data[13].max := 1.0, [71].log_data[13].total := 3600.0, [71].log_data[13].time := 3600.0, [71].log_data[13].valid := 1, [71].log_data[14].time := 3600.0, [71].log_data[14].valid := 1, [71].log_data[15].time := 3600.0, [71].log_data[15].valid := 1, [71].log_data[16].time := 3600.0, [71].log_data[16].valid := 1, [71].log_data[17].min := 1.0, [71].log_data[17].max := 1.0, [71].log_data[17].total := 3600.0, [71].log_data[17].time := 3600.0, [71].log_data[17].valid := 1, [71].log_data[18].time := 3600.0, [71].log_data[18].valid := 1, [71].log_data[19].time := 3600.0, [71].log_data[19].valid := 1, [71].log_data[20].time := 3600.0, [71].log_data[20].valid := 1, [71].log_data[21].min := 1.0, [71].log_data[21].max := 1.0, [71].log_data[21].total := 3600.0, [71].log_data[21].time := 3600.0, [71].log_data[21].valid := 1, [71].log_data[22].time := 3600.0, [71].log_data[22].valid := 1, [71].log_data[23].time := 3600.0, [71].log_data[23].valid := 1, [71].log_data[24].time := 3600.0, [71].log_data[24].valid := 1, [71].log_data[25].time := 3600.0, [71].log_data[25].valid := 1, [71].log_data[26].time := 3600.0, [71].log_data[26].valid := 1, [71].log_data[27].time := 3600.0, [71].log_data[27].valid := 1, [71].log_data[28].time := 3600.0, [71].log_data[28].valid := 1, [71].log_data[29].min := 1.0, [71].log_data[29].max := 1.0, [71].log_data[29].total := 3600.0, [71].log_data[29].time := 3600.0, [71].log_data[29].valid := 1, [71].log_data[30].min := 1.0, [71].log_data[30].max := 1.0, [71].log_data[30].total := 3600.0, [71].log_data[30].time := 3600.0, [71].log_data[30].valid := 1,
        [71].log_data[31].max := 1.0, [71].log_data[31].total := 1440.998, [71].log_data[31].time := 3600.0, [71].log_data[31].valid := 1, [71].log_data[32].max := 1.0, [71].log_data[32].total := 1629.998, [71].log_data[32].time := 3600.0, [71].log_data[32].maxminute := 2, [71].log_data[32].valid := 1, [71].log_data[33].time := 3600.0, [71].log_data[33].valid := 1, [71].log_data[34].time := 3600.0, [71].log_data[34].valid := 1, [71].log_data[35].max := 1.0, [71].log_data[35].total := 1440.7471, [71].log_data[35].time := 3600.0, [71].log_data[35].minminute := 4, [71].log_data[35].valid := 1, [71].log_data[36].max := 1.0, [71].log_data[36].total := 1629.7471, [71].log_data[36].time := 3600.0, [71].log_data[36].maxminute := 6, [71].log_data[36].valid := 1, [71].log_data[37].max := 7.5763884, [71].log_data[37].total := 3403.9104, [71].log_data[37].time := 3600.0, [71].log_data[37].maxminute := 47, [71].log_data[37].valid := 1, [71].log_data[38].time := 3600.0, [71].log_data[38].valid := 1, [71].log_data[39].min := 0.99494183, [71].log_data[39].max := 1.0216767, [71].log_data[39].total := 3610.9382, [71].log_data[39].time := 3600.0, [71].log_data[39].minminute := 28, [71].log_data[39].maxminute := 48, [71].log_data[39].valid := 1, [71].log_data[40].min := 7.555797, [71].log_data[40].max := 7.6060877, [71].log_data[40].total := 27330.9, [71].log_data[40].time := 3600.0, [71].log_data[40].minminute := 55, [71].log_data[40].maxminute := 49, [71].log_data[40].valid := 1, [71].log_data[41].min := 0.022540038, [71].log_data[41].max := 0.037261963, [71].log_data[41].total := 100.76825, [71].log_data[41].time := 3600.0, [71].log_data[41].minminute := 40, [71].log_data[41].maxminute := 10, [71].log_data[41].valid := 1, [71].log_data[42].min := 2.291996, [71].log_data[42].max := 2.2964714, [71].log_data[42].total := 8259.494, [71].log_data[42].time := 3600.0, [71].log_data[42].minminute := 6, [71].log_data[42].maxminute := 11, [71].log_data[42].valid := 1, [71].log_data[43].min := -0.27999878, [71].log_data[43].max := -0.26000214,
        [71].log_data[43].total := -991.07214, [71].log_data[43].time := 3600.0, [71].log_data[43].valid := 1, [71].log_data[44].min := -0.3199997, [71].log_data[44].max := -0.30000305, [71].log_data[44].total := -1080.0961, [71].log_data[44].time := 3600.0, [71].log_data[44].minminute := 1, [71].log_data[44].valid := 1, [71].log_data[45].time := 3600.0, [71].log_data[45].valid := 1, [71].log_data[46].time := 3600.0, [71].log_data[46].valid := 1, [71].log_data[47].time := 3600.0, [71].log_data[47].valid := 1, [71].log_data[48].min := 6.761053, [71].log_data[48].max := 6.9748535, [71].log_data[48].total := 24439.693, [71].log_data[48].time := 3600.0, [71].log_data[48].minminute := 59, [71].log_data[48].maxminute := 54, [71].log_data[48].valid := 1, [71].log_data[49].min := 7.9570303, [71].log_data[49].max := 9.80001, [71].log_data[49].total := 34550.37, [71].log_data[49].time := 3600.0, [71].log_data[49].minminute := 59, [71].log_data[49].maxminute := 14, [71].log_data[49].valid := 1, [71].log_data[50].min := 2.1061473, [71].log_data[50].max := 2.2070804, [71].log_data[50].total := 7742.4414, [71].log_data[50].time := 3600.0, [71].log_data[50].minminute := 48, [71].log_data[50].maxminute := 56, [71].log_data[50].valid := 1, [71].log_data[51].time := 3600.0, [71].log_data[51].valid := 1, [71].log_data[52].min := -3.1200027, [71].log_data[52].max := 0.11999512, [71].log_data[52].total := -7864.1772, [71].log_data[52].time := 3600.0, [71].log_data[52].minminute := 23, [71].log_data[52].valid := 1, [71].log_data[53].min := -2.600006, [71].log_data[53].max := 0.27999878, [71].log_data[53].total := -7363.315, [71].log_data[53].time := 3600.0, [71].log_data[53].minminute := 17, [71].log_data[53].maxminute := 37, [71].log_data[53].valid := 1, [71].log_data[54].max := 0.5585, [71].log_data[54].total := 1217.4135, [71].log_data[54].time := 3600.0, [71].log_data[54].maxminute := 23, [71].log_data[54].valid := 1, [71].log_data[55].max := 0.543, [71].log_data[55].total := 1217.2546, [71].log_data[55].time := 3600.0, [71].log_data[55].minminute := 4,
        [71].log_data[55].maxminute := 6, [71].log_data[55].valid := 1, [71].log_data[56].min := 0.16004932, [71].log_data[56].max := 0.16055967, [71].log_data[56].total := 576.91345, [71].log_data[56].time := 3600.0, [71].log_data[56].maxminute := 36, [71].log_data[56].valid := 1, [71].log_data[57].min := 0.25733134, [71].log_data[57].max := 0.25776318, [71].log_data[57].total := 927.0978, [71].log_data[57].time := 3600.0, [71].log_data[57].minminute := 20, [71].log_data[57].maxminute := 30, [71].log_data[57].valid := 1, [71].log_data[58].time := 3600.0, [71].log_data[58].valid := 1, [71].log_data[59].time := 3600.0, [71].log_data[59].valid := 1, [71].log_data[60].valid := 1, [71].log_data[61].valid := 1, [71].log_data[62].valid := 1, [71].log_data[63].valid := 1, [71].log_data[64].valid := 1, [71].log_data[65].valid := 1, [71].log_data[66].valid := 1, [71].log_data[67].valid := 1, [71].log_data[68].valid := 1, [71].log_data[69].valid := 1, [71].log_data[70].valid := 1, [71].log_data[71].valid := 1, [71].log_data[72].valid := 1, [71].log_data[73].valid := 1, [71].log_data[74].valid := 1, [71].log_data[75].valid := 1, [71].log_data[76].valid := 1, [71].log_data[77].valid := 1, [71].log_data[78].valid := 1, [71].log_data[79].valid := 1, [71].log_data[80].valid := 1, [71].log_data[81].valid := 1, [71].log_data[82].valid := 1, [71].log_data[83].valid := 1, [71].log_data[84].valid := 1, [71].log_data[85].valid := 1, [71].log_data[86].valid := 1, [71].log_data[87].valid := 1, [71].log_data[88].valid := 1, [71].log_data[89].valid := 1, [71].log_data[90].valid := 1, [71].log_data[91].valid := 1, [71].log_data[92].valid := 1, [71].log_data[93].valid := 1, [71].log_data[94].valid := 1, [71].log_data[95].valid := 1, [71].log_data[96].valid := 1, [71].log_data[97].valid := 1, [71].log_data[98].valid := 1, [71].log_data[99].valid := 1, [71].log_data[100].valid := 1,
        [71].log_data[101].valid := 1, [71].log_data[102].valid := 1, [71].log_data[103].valid := 1, [71].log_data[104].valid := 1, [71].log_data[105].valid := 1, [71].log_data[106].valid := 1, [71].log_data[107].valid := 1, [71].log_data[108].valid := 1, [71].log_data[109].valid := 1, [71].log_data[110].valid := 1, [71].log_data[111].valid := 1, [71].log_data[112].valid := 1, [71].log_data[113].valid := 1, [71].log_data[114].valid := 1, [71].log_data[115].valid := 1, [71].log_data[116].valid := 1, [71].log_data[117].valid := 1, [71].log_data[118].valid := 1, [71].log_data[119].valid := 1, [71].log_data[120].valid := 1, [71].log_data[121].valid := 1, [71].log_data[122].valid := 1, [71].log_data[123].valid := 1, [71].log_data[124].valid := 1, [71].time.Year := 2023, [71].time.Month := 1, [71].time.Day := 16, [71].time.Hour := 2, [71].time.Minute := 59, [71].time.Second := 59, [72].log_data[0].min := 1.0, [72].log_data[0].max := 1.0, [72].log_data[0].total := 3600.0, [72].log_data[0].time := 3600.0, [72].log_data[0].valid := 1, [72].log_data[1].time := 3600.0, [72].log_data[1].valid := 1, [72].log_data[2].time := 3600.0, [72].log_data[2].valid := 1, [72].log_data[3].time := 3600.0, [72].log_data[3].valid := 1, [72].log_data[4].time := 3600.0, [72].log_data[4].valid := 1, [72].log_data[5].time := 3600.0, [72].log_data[5].valid := 1, [72].log_data[6].time := 3600.0, [72].log_data[6].valid := 1, [72].log_data[7].time := 3600.0, [72].log_data[7].valid := 1, [72].log_data[8].min := 1.0, [72].log_data[8].max := 1.0, [72].log_data[8].total := 3600.0, [72].log_data[8].time := 3600.0, [72].log_data[8].valid := 1, [72].log_data[9].min := 1.0, [72].log_data[9].max := 1.0, [72].log_data[9].total := 3600.0, [72].log_data[9].time := 3600.0, [72].log_data[9].valid := 1, [72].log_data[10].min := 1.0,
        [72].log_data[10].max := 1.0, [72].log_data[10].total := 3600.0, [72].log_data[10].time := 3600.0, [72].log_data[10].valid := 1, [72].log_data[11].time := 3600.0, [72].log_data[11].valid := 1, [72].log_data[12].min := 1.0, [72].log_data[12].max := 1.0, [72].log_data[12].total := 3600.0, [72].log_data[12].time := 3600.0, [72].log_data[12].valid := 1, [72].log_data[13].min := 1.0, [72].log_data[13].max := 1.0, [72].log_data[13].total := 3600.0, [72].log_data[13].time := 3600.0, [72].log_data[13].valid := 1, [72].log_data[14].time := 3600.0, [72].log_data[14].valid := 1, [72].log_data[15].time := 3600.0, [72].log_data[15].valid := 1, [72].log_data[16].time := 3600.0, [72].log_data[16].valid := 1, [72].log_data[17].min := 1.0, [72].log_data[17].max := 1.0, [72].log_data[17].total := 3600.0, [72].log_data[17].time := 3600.0, [72].log_data[17].valid := 1, [72].log_data[18].time := 3600.0, [72].log_data[18].valid := 1, [72].log_data[19].time := 3600.0, [72].log_data[19].valid := 1, [72].log_data[20].time := 3600.0, [72].log_data[20].valid := 1, [72].log_data[21].min := 1.0, [72].log_data[21].max := 1.0, [72].log_data[21].total := 3600.0, [72].log_data[21].time := 3600.0, [72].log_data[21].valid := 1, [72].log_data[22].time := 3600.0, [72].log_data[22].valid := 1, [72].log_data[23].time := 3600.0, [72].log_data[23].valid := 1, [72].log_data[24].time := 3600.0, [72].log_data[24].valid := 1, [72].log_data[25].time := 3600.0, [72].log_data[25].valid := 1, [72].log_data[26].time := 3600.0, [72].log_data[26].valid := 1, [72].log_data[27].time := 3600.0, [72].log_data[27].valid := 1, [72].log_data[28].time := 3600.0, [72].log_data[28].valid := 1, [72].log_data[29].min := 1.0, [72].log_data[29].max := 1.0, [72].log_data[29].total := 3600.0, [72].log_data[29].time := 3600.0, [72].log_data[29].valid := 1, [72].log_data[30].min := 1.0, [72].log_data[30].max := 1.0, [72].log_data[30].total := 3600.0,
        [72].log_data[30].time := 3600.0, [72].log_data[30].valid := 1, [72].log_data[31].max := 1.0, [72].log_data[31].total := 1440.7471, [72].log_data[31].time := 3600.0, [72].log_data[31].minminute := 3, [72].log_data[31].valid := 1, [72].log_data[32].max := 1.0, [72].log_data[32].total := 1629.998, [72].log_data[32].time := 3600.0, [72].log_data[32].maxminute := 5, [72].log_data[32].valid := 1, [72].log_data[33].time := 3600.0, [72].log_data[33].valid := 1, [72].log_data[34].time := 3600.0, [72].log_data[34].valid := 1, [72].log_data[35].max := 1.0, [72].log_data[35].total := 1553.498, [72].log_data[35].time := 3600.0, [72].log_data[35].minminute := 7, [72].log_data[35].valid := 1, [72].log_data[36].max := 1.0, [72].log_data[36].total := 1605.2471, [72].log_data[36].time := 3600.0, [72].log_data[36].maxminute := 9, [72].log_data[36].valid := 1, [72].log_data[37].time := 3600.0, [72].log_data[37].valid := 1, [72].log_data[38].time := 3600.0, [72].log_data[38].valid := 1, [72].log_data[39].min := 0.99623734, [72].log_data[39].max := 1.0067194, [72].log_data[39].total := 3607.0427, [72].log_data[39].time := 3600.0, [72].log_data[39].minminute := 26, [72].log_data[39].maxminute := 31, [72].log_data[39].valid := 1, [72].log_data[40].min := 7.574485, [72].log_data[40].max := 7.6063623, [72].log_data[40].total := 27328.861, [72].log_data[40].time := 3600.0, [72].log_data[40].minminute := 7, [72].log_data[40].maxminute := 36, [72].log_data[40].valid := 1, [72].log_data[41].min := 0.022540038, [72].log_data[41].max := 0.026073486, [72].log_data[41].total := 82.99852, [72].log_data[41].time := 3600.0, [72].log_data[41].minminute := 1, [72].log_data[41].maxminute := 31, [72].log_data[41].valid := 1, [72].log_data[42].min := 2.2918782, [72].log_data[42].max := 2.296236, [72].log_data[42].total := 8259.391, [72].log_data[42].time := 3600.0, [72].log_data[42].minminute := 33, [72].log_data[42].maxminute := 1, [72].log_data[42].valid := 1, [72].log_data[43].min := -0.27999878, [72].log_data[43].max := -0.26000214,
